MoveL Offs(p0,294.46809999999994,373.47709999999995, 0), v100, z5, tool0;
MoveL Offs(p0,293.07520000000005,371.8112, 0), v100, z5, tool0;
MoveL Offs(p0,291.8875,370.5125, 0), v100, z5, tool0;
MoveL Offs(p0,290.8528,369.5288, 0), v100, z5, tool0;
MoveL Offs(p0,289.9189,368.80789999999996, 0), v100, z5, tool0;
MoveL Offs(p0,289.03360000000004,368.29760000000005, 0), v100, z5, tool0;
MoveL Offs(p0,288.1447,367.94570000000004, 0), v100, z5, tool0;
MoveL Offs(p0,287.2,367.7, 0), v100, z5, tool0;
MoveL Offs(p0,283.18910000000005,366.95770000000005, 0), v100, z5, tool0;
MoveL Offs(p0,279.59280000000007,366.4176000000001, 0), v100, z5, tool0;
MoveL Offs(p0,276.28569999999996,366.08990000000006, 0), v100, z5, tool0;
MoveL Offs(p0,273.1424,365.9848, 0), v100, z5, tool0;
MoveL Offs(p0,270.0375,366.1125, 0), v100, z5, tool0;
MoveL Offs(p0,266.8456,366.4832, 0), v100, z5, tool0;
MoveL Offs(p0,263.4413,367.1071, 0), v100, z5, tool0;
MoveL Offs(p0,259.6992,367.99440000000004, 0), v100, z5, tool0;
MoveL Offs(p0,255.49390000000002,369.1553, 0), v100, z5, tool0;
MoveL Offs(p0,250.7,370.6, 0), v100, z5, tool0;
MoveL Offs(p0,248.47970000000004,371.28720000000004, 0), v100, z5, tool0;
MoveL Offs(p0,246.31760000000008,371.90960000000007, 0), v100, z5, tool0;
MoveL Offs(p0,244.21189999999996,372.4684, 0), v100, z5, tool0;
MoveL Offs(p0,242.16079999999997,372.9648, 0), v100, z5, tool0;
MoveL Offs(p0,240.1625,373.4, 0), v100, z5, tool0;
MoveL Offs(p0,238.2152,373.7752, 0), v100, z5, tool0;
MoveL Offs(p0,236.31709999999998,374.0916, 0), v100, z5, tool0;
MoveL Offs(p0,234.46640000000002,374.35040000000004, 0), v100, z5, tool0;
MoveL Offs(p0,232.66130000000004,374.55280000000005, 0), v100, z5, tool0;
MoveL Offs(p0,230.9,374.7, 0), v100, z5, tool0;
MoveL Offs(p0,222.3,375.3, 0), v100, z5, tool0;
MoveL Offs(p0,221.6,384.4, 0), v100, z5, tool0;
MoveL Offs(p0,221.27370000000005,388.0507, 0), v100, z5, tool0;
MoveL Offs(p0,220.78960000000006,392.02960000000013, 0), v100, z5, tool0;
MoveL Offs(p0,220.1699,396.22690000000006, 0), v100, z5, tool0;
MoveL Offs(p0,219.43680000000003,400.53280000000007, 0), v100, z5, tool0;
MoveL Offs(p0,218.6125,404.8375, 0), v100, z5, tool0;
MoveL Offs(p0,217.7192,409.0312, 0), v100, z5, tool0;
MoveL Offs(p0,216.77910000000003,413.0041, 0), v100, z5, tool0;
MoveL Offs(p0,215.81440000000003,416.6464000000001, 0), v100, z5, tool0;
MoveL Offs(p0,214.8473,419.8483, 0), v100, z5, tool0;
MoveL Offs(p0,213.9,422.5, 0), v100, z5, tool0;
MoveL Offs(p0,213.26730000000003,424.0777, 0), v100, z5, tool0;
MoveL Offs(p0,212.72640000000007,425.3536000000002, 0), v100, z5, tool0;
MoveL Offs(p0,212.2431,426.3619, 0), v100, z5, tool0;
MoveL Offs(p0,211.78320000000002,427.13680000000005, 0), v100, z5, tool0;
MoveL Offs(p0,211.3125,427.7125, 0), v100, z5, tool0;
MoveL Offs(p0,210.7968,428.1232, 0), v100, z5, tool0;
MoveL Offs(p0,210.20190000000002,428.4031, 0), v100, z5, tool0;
MoveL Offs(p0,209.49360000000001,428.5864, 0), v100, z5, tool0;
MoveL Offs(p0,208.6377,428.70730000000003, 0), v100, z5, tool0;
MoveL Offs(p0,207.6,428.8, 0), v100, z5, tool0;
MoveL Offs(p0,203.7,429.1, 0), v100, z5, tool0;
MoveL Offs(p0,204.4,419.3, 0), v100, z5, tool0;
MoveL Offs(p0,205.0,409.5, 0), v100, z5, tool0;
MoveL Offs(p0,201.9,417.0, 0), v100, z5, tool0;
MoveL Offs(p0,200.11920000000003,421.2125000000001, 0), v100, z5, tool0;
MoveL Offs(p0,198.11760000000004,425.7280000000002, 0), v100, z5, tool0;
MoveL Offs(p0,195.9564,430.4235, 0), v100, z5, tool0;
MoveL Offs(p0,193.69680000000002,435.17600000000004, 0), v100, z5, tool0;
MoveL Offs(p0,191.4,439.8625, 0), v100, z5, tool0;
MoveL Offs(p0,189.1272,444.36, 0), v100, z5, tool0;
MoveL Offs(p0,186.9396,448.5455, 0), v100, z5, tool0;
MoveL Offs(p0,184.8984,452.2960000000001, 0), v100, z5, tool0;
MoveL Offs(p0,183.06480000000002,455.48850000000004, 0), v100, z5, tool0;
MoveL Offs(p0,181.5,458.0, 0), v100, z5, tool0;
MoveL Offs(p0,179.79570000000004,460.49500000000006, 0), v100, z5, tool0;
MoveL Offs(p0,178.25760000000002,462.6000000000002, 0), v100, z5, tool0;
MoveL Offs(p0,176.8479,464.34499999999997, 0), v100, z5, tool0;
MoveL Offs(p0,175.5288,465.76000000000005, 0), v100, z5, tool0;
MoveL Offs(p0,174.2625,466.875, 0), v100, z5, tool0;
MoveL Offs(p0,173.0112,467.71999999999997, 0), v100, z5, tool0;
MoveL Offs(p0,171.7371,468.325, 0), v100, z5, tool0;
MoveL Offs(p0,170.4024,468.7200000000001, 0), v100, z5, tool0;
MoveL Offs(p0,168.96930000000003,468.93500000000006, 0), v100, z5, tool0;
MoveL Offs(p0,167.4,469.0, 0), v100, z5, tool0;
MoveL Offs(p0,164.1664,468.7728000000001, 0), v100, z5, tool0;
MoveL Offs(p0,163.7375,468.6125, 0), v100, z5, tool0;
MoveL Offs(p0,163.4256,468.39519999999993, 0), v100, z5, tool0;
MoveL Offs(p0,163.2133,468.11310000000003, 0), v100, z5, tool0;
MoveL Offs(p0,163.0832,467.75840000000005, 0), v100, z5, tool0;
MoveL Offs(p0,163.0179,467.3233, 0), v100, z5, tool0;
MoveL Offs(p0,163.0,466.8, 0), v100, z5, tool0;
MoveL Offs(p0,163.0,466.8, 0), v100, z5, tool0;
MoveJ Offs(p0,173.0,464.5, 10), v100, z1, tool0;
MoveL Offs(p0,174.1694,463.2745000000001, 0), v100, z5, tool0;
MoveL Offs(p0,175.55120000000005,461.56000000000023, 0), v100, z5, tool0;
MoveL Offs(p0,177.1058,459.41949999999997, 0), v100, z5, tool0;
MoveL Offs(p0,178.79360000000003,456.916, 0), v100, z5, tool0;
MoveL Offs(p0,180.575,454.1125, 0), v100, z5, tool0;
MoveL Offs(p0,182.4104,451.07199999999995, 0), v100, z5, tool0;
MoveL Offs(p0,184.2602,447.8575000000001, 0), v100, z5, tool0;
MoveL Offs(p0,186.08480000000003,444.532, 0), v100, z5, tool0;
MoveL Offs(p0,187.8446,441.1585, 0), v100, z5, tool0;
MoveL Offs(p0,189.5,437.8, 0), v100, z5, tool0;
MoveL Offs(p0,191.66320000000002,433.08140000000003, 0), v100, z5, tool0;
MoveL Offs(p0,193.79760000000005,428.1432000000001, 0), v100, z5, tool0;
MoveL Offs(p0,195.85039999999998,423.1318, 0), v100, z5, tool0;
MoveL Offs(p0,197.7688,418.19360000000006, 0), v100, z5, tool0;
MoveL Offs(p0,199.5,413.475, 0), v100, z5, tool0;
MoveL Offs(p0,200.9912,409.1224, 0), v100, z5, tool0;
MoveL Offs(p0,202.1896,405.2822, 0), v100, z5, tool0;
MoveL Offs(p0,203.04240000000001,402.10080000000005, 0), v100, z5, tool0;
MoveL Offs(p0,203.4968,399.7246, 0), v100, z5, tool0;
MoveL Offs(p0,203.5,398.3, 0), v100, z5, tool0;
MoveL Offs(p0,203.88400000000001,396.0856, 0), v100, z5, tool0;
MoveL Offs(p0,204.121,396.0212, 0), v100, z5, tool0;
MoveL Offs(p0,204.4,396.0, 0), v100, z5, tool0;
MoveL Offs(p0,205.57200000000006,396.43520000000007, 0), v100, z5, tool0;
MoveL Offs(p0,206.01099999999997,397.05029999999994, 0), v100, z5, tool0;
MoveL Offs(p0,206.36000000000004,397.9936, 0), v100, z5, tool0;
MoveL Offs(p0,206.625,399.3125, 0), v100, z5, tool0;
MoveL Offs(p0,206.81199999999998,401.0544, 0), v100, z5, tool0;
MoveL Offs(p0,206.927,403.2667, 0), v100, z5, tool0;
MoveL Offs(p0,206.97600000000003,405.9968, 0), v100, z5, tool0;
MoveL Offs(p0,206.965,409.2921, 0), v100, z5, tool0;
MoveL Offs(p0,206.9,413.2, 0), v100, z5, tool0;
MoveL Offs(p0,207.1384,424.5264000000001, 0), v100, z5, tool0;
MoveL Offs(p0,207.4125,425.8625, 0), v100, z5, tool0;
MoveL Offs(p0,207.78560000000002,426.6496, 0), v100, z5, tool0;
MoveL Offs(p0,208.2643,426.91229999999996, 0), v100, z5, tool0;
MoveL Offs(p0,208.85520000000002,426.6752, 0), v100, z5, tool0;
MoveL Offs(p0,209.56490000000002,425.9629, 0), v100, z5, tool0;
MoveL Offs(p0,210.4,424.8, 0), v100, z5, tool0;
MoveL Offs(p0,211.00590000000003,423.62250000000006, 0), v100, z5, tool0;
MoveL Offs(p0,211.67120000000006,421.8840000000001, 0), v100, z5, tool0;
MoveL Offs(p0,212.37730000000002,419.66549999999995, 0), v100, z5, tool0;
MoveL Offs(p0,213.1056,417.04799999999994, 0), v100, z5, tool0;
MoveL Offs(p0,213.8375,414.1125, 0), v100, z5, tool0;
MoveL Offs(p0,214.55440000000004,410.93999999999994, 0), v100, z5, tool0;
MoveL Offs(p0,215.2377,407.6115, 0), v100, z5, tool0;
MoveL Offs(p0,215.86880000000002,404.208, 0), v100, z5, tool0;
MoveL Offs(p0,216.4291,400.81050000000005, 0), v100, z5, tool0;
MoveL Offs(p0,216.9,397.5, 0), v100, z5, tool0;
MoveL Offs(p0,217.40370000000001,393.5277000000001, 0), v100, z5, tool0;
MoveL Offs(p0,217.83360000000008,389.8536000000001, 0), v100, z5, tool0;
MoveL Offs(p0,218.18789999999998,386.51189999999997, 0), v100, z5, tool0;
MoveL Offs(p0,218.46480000000003,383.5368, 0), v100, z5, tool0;
MoveL Offs(p0,218.6625,380.9625, 0), v100, z5, tool0;
MoveL Offs(p0,218.7792,378.8232, 0), v100, z5, tool0;
MoveL Offs(p0,218.8131,377.1531, 0), v100, z5, tool0;
MoveL Offs(p0,218.7624,375.98640000000006, 0), v100, z5, tool0;
MoveL Offs(p0,218.6253,375.3573, 0), v100, z5, tool0;
MoveL Offs(p0,218.4,375.3, 0), v100, z5, tool0;
MoveL Offs(p0,218.07510000000002,375.6689, 0), v100, z5, tool0;
MoveL Offs(p0,217.42080000000004,376.45120000000014, 0), v100, z5, tool0;
MoveL Offs(p0,216.46769999999998,377.6103, 0), v100, z5, tool0;
MoveL Offs(p0,215.24640000000005,379.10960000000006, 0), v100, z5, tool0;
MoveL Offs(p0,213.7875,380.9125, 0), v100, z5, tool0;
MoveL Offs(p0,212.1216,382.9824, 0), v100, z5, tool0;
MoveL Offs(p0,210.2793,385.28270000000003, 0), v100, z5, tool0;
MoveL Offs(p0,208.29120000000003,387.77680000000004, 0), v100, z5, tool0;
MoveL Offs(p0,206.18789999999998,390.4281, 0), v100, z5, tool0;
MoveL Offs(p0,204.0,393.2, 0), v100, z5, tool0;
MoveL Offs(p0,201.8005,396.0019000000001, 0), v100, z5, tool0;
MoveL Offs(p0,199.66400000000004,398.68320000000006, 0), v100, z5, tool0;
MoveL Offs(p0,197.62349999999998,401.2073, 0), v100, z5, tool0;
MoveL Offs(p0,195.71200000000002,403.5376, 0), v100, z5, tool0;
MoveL Offs(p0,193.9625,405.6375, 0), v100, z5, tool0;
MoveL Offs(p0,192.40800000000002,407.4704, 0), v100, z5, tool0;
MoveL Offs(p0,191.0815,408.99969999999996, 0), v100, z5, tool0;
MoveL Offs(p0,190.01600000000002,410.1888, 0), v100, z5, tool0;
MoveL Offs(p0,189.24450000000002,411.00110000000006, 0), v100, z5, tool0;
MoveL Offs(p0,188.8,411.4, 0), v100, z5, tool0;
MoveL Offs(p0,188.18900000000002,411.6944, 0), v100, z5, tool0;
MoveL Offs(p0,187.56000000000003,411.85920000000004, 0), v100, z5, tool0;
MoveL Offs(p0,186.919,411.8968, 0), v100, z5, tool0;
MoveL Offs(p0,186.27200000000002,411.80959999999993, 0), v100, z5, tool0;
MoveL Offs(p0,185.625,411.6, 0), v100, z5, tool0;
MoveL Offs(p0,184.35499999999996,410.8232, 0), v100, z5, tool0;
MoveL Offs(p0,183.744,410.2608, 0), v100, z5, tool0;
MoveL Offs(p0,183.157,409.5856, 0), v100, z5, tool0;
MoveL Offs(p0,182.6,408.8, 0), v100, z5, tool0;
MoveL Offs(p0,182.29110000000003,408.22150000000005, 0), v100, z5, tool0;
MoveL Offs(p0,182.14480000000006,407.54400000000015, 0), v100, z5, tool0;
MoveL Offs(p0,182.2517,406.55449999999996, 0), v100, z5, tool0;
MoveL Offs(p0,183.5875,402.7875, 0), v100, z5, tool0;
MoveL Offs(p0,184.9976,399.58399999999995, 0), v100, z5, tool0;
MoveL Offs(p0,187.0233,395.2165, 0), v100, z5, tool0;
MoveL Offs(p0,189.7552,389.47200000000004, 0), v100, z5, tool0;
MoveL Offs(p0,193.28390000000002,382.1375, 0), v100, z5, tool0;
MoveL Offs(p0,197.7,373.0, 0), v100, z5, tool0;
MoveL Offs(p0,199.66400000000002,368.88100000000014, 0), v100, z5, tool0;
MoveL Offs(p0,201.52000000000007,364.96000000000004, 0), v100, z5, tool0;
MoveL Offs(p0,203.244,361.29100000000005, 0), v100, z5, tool0;
MoveL Offs(p0,204.81200000000004,357.928, 0), v100, z5, tool0;
MoveL Offs(p0,206.2,354.925, 0), v100, z5, tool0;
MoveL Offs(p0,207.38400000000001,352.33599999999996, 0), v100, z5, tool0;
MoveL Offs(p0,208.34,350.21500000000003, 0), v100, z5, tool0;
MoveL Offs(p0,209.04400000000004,348.61600000000004, 0), v100, z5, tool0;
MoveL Offs(p0,209.47200000000004,347.593, 0), v100, z5, tool0;
MoveL Offs(p0,209.6,347.2, 0), v100, z5, tool0;
MoveL Offs(p0,208.92859999999996,347.4196, 0), v100, z5, tool0;
MoveL Offs(p0,208.5152,347.6512000000001, 0), v100, z5, tool0;
MoveL Offs(p0,208.025,347.95, 0), v100, z5, tool0;
MoveL Offs(p0,207.46880000000002,348.3088, 0), v100, z5, tool0;
MoveL Offs(p0,206.85739999999996,348.7204, 0), v100, z5, tool0;
MoveL Offs(p0,206.2016,349.17760000000004, 0), v100, z5, tool0;
MoveL Offs(p0,205.51220000000004,349.67320000000007, 0), v100, z5, tool0;
MoveL Offs(p0,204.8,350.2, 0), v100, z5, tool0;
MoveL Offs(p0,203.59520000000003,351.0874, 0), v100, z5, tool0;
MoveL Offs(p0,202.32560000000007,351.9472000000001, 0), v100, z5, tool0;
MoveL Offs(p0,200.9984,352.7758, 0), v100, z5, tool0;
MoveL Offs(p0,199.62080000000003,353.5696, 0), v100, z5, tool0;
MoveL Offs(p0,198.2,354.325, 0), v100, z5, tool0;
MoveL Offs(p0,196.7432,355.0384, 0), v100, z5, tool0;
MoveL Offs(p0,195.2576,355.70619999999997, 0), v100, z5, tool0;
MoveL Offs(p0,193.75040000000004,356.3248, 0), v100, z5, tool0;
MoveL Offs(p0,192.2288,356.8906, 0), v100, z5, tool0;
MoveL Offs(p0,190.7,357.4, 0), v100, z5, tool0;
MoveL Offs(p0,190.04080000000005,357.8960000000001, 0), v100, z5, tool0;
MoveL Offs(p0,189.63619999999997,358.3585, 0), v100, z5, tool0;
MoveL Offs(p0,189.1944,358.944, 0), v100, z5, tool0;
MoveL Offs(p0,188.725,359.6375, 0), v100, z5, tool0;
MoveL Offs(p0,188.2376,360.424, 0), v100, z5, tool0;
MoveL Offs(p0,187.7418,361.2885, 0), v100, z5, tool0;
MoveL Offs(p0,187.24720000000002,362.216, 0), v100, z5, tool0;
MoveL Offs(p0,186.7634,363.1915, 0), v100, z5, tool0;
MoveL Offs(p0,186.3,364.2, 0), v100, z5, tool0;
MoveL Offs(p0,185.02380000000002,367.0821, 0), v100, z5, tool0;
MoveL Offs(p0,183.65040000000005,370.0368000000001, 0), v100, z5, tool0;
MoveL Offs(p0,182.1726,373.07669999999996, 0), v100, z5, tool0;
MoveL Offs(p0,180.58319999999998,376.2144, 0), v100, z5, tool0;
MoveL Offs(p0,178.875,379.4625, 0), v100, z5, tool0;
MoveL Offs(p0,177.04080000000002,382.83360000000005, 0), v100, z5, tool0;
MoveL Offs(p0,175.0734,386.3403, 0), v100, z5, tool0;
MoveL Offs(p0,172.96560000000002,389.9952, 0), v100, z5, tool0;
MoveL Offs(p0,170.71020000000001,393.81090000000006, 0), v100, z5, tool0;
MoveL Offs(p0,168.3,397.8, 0), v100, z5, tool0;
MoveL Offs(p0,167.0781,399.8056, 0), v100, z5, tool0;
MoveL Offs(p0,165.94080000000005,401.7248000000001, 0), v100, z5, tool0;
MoveL Offs(p0,164.90069999999997,403.5312, 0), v100, z5, tool0;
MoveL Offs(p0,163.9704,405.19840000000005, 0), v100, z5, tool0;
MoveL Offs(p0,163.1625,406.7, 0), v100, z5, tool0;
MoveL Offs(p0,162.48960000000002,408.0096, 0), v100, z5, tool0;
MoveL Offs(p0,161.9643,409.1008, 0), v100, z5, tool0;
MoveL Offs(p0,161.59920000000002,409.94719999999995, 0), v100, z5, tool0;
MoveL Offs(p0,161.4069,410.5224, 0), v100, z5, tool0;
MoveL Offs(p0,161.4,410.8, 0), v100, z5, tool0;
MoveL Offs(p0,163.78140000000002,410.3509, 0), v100, z5, tool0;
MoveL Offs(p0,165.0688,409.7888000000001, 0), v100, z5, tool0;
MoveL Offs(p0,166.475,409.0875, 0), v100, z5, tool0;
MoveL Offs(p0,167.9232,408.2872, 0), v100, z5, tool0;
MoveL Offs(p0,169.3366,407.4281, 0), v100, z5, tool0;
MoveL Offs(p0,170.6384,406.5504, 0), v100, z5, tool0;
MoveL Offs(p0,171.7518,405.6943, 0), v100, z5, tool0;
MoveL Offs(p0,172.6,404.9, 0), v100, z5, tool0;
MoveL Offs(p0,172.97840000000002,404.47540000000004, 0), v100, z5, tool0;
MoveL Offs(p0,173.2752,404.0952000000001, 0), v100, z5, tool0;
MoveL Offs(p0,173.4928,403.7498, 0), v100, z5, tool0;
MoveL Offs(p0,173.63360000000003,403.42960000000005, 0), v100, z5, tool0;
MoveL Offs(p0,173.7,403.125, 0), v100, z5, tool0;
MoveL Offs(p0,173.6944,402.82640000000004, 0), v100, z5, tool0;
MoveL Offs(p0,173.6192,402.5242, 0), v100, z5, tool0;
MoveL Offs(p0,173.4768,402.2088, 0), v100, z5, tool0;
MoveL Offs(p0,173.2696,401.8706, 0), v100, z5, tool0;
MoveL Offs(p0,173.0,401.5, 0), v100, z5, tool0;
MoveL Offs(p0,172.70970000000003,401.1421, 0), v100, z5, tool0;
MoveL Offs(p0,172.50160000000005,400.8448000000001, 0), v100, z5, tool0;
MoveL Offs(p0,172.37989999999996,400.6027, 0), v100, z5, tool0;
MoveL Offs(p0,172.34880000000004,400.41040000000004, 0), v100, z5, tool0;
MoveL Offs(p0,172.4125,400.2625, 0), v100, z5, tool0;
MoveL Offs(p0,172.5752,400.1536, 0), v100, z5, tool0;
MoveL Offs(p0,173.2144,400.0312, 0), v100, z5, tool0;
MoveL Offs(p0,173.6993,400.00690000000003, 0), v100, z5, tool0;
MoveL Offs(p0,174.3,400.0, 0), v100, z5, tool0;
MoveL Offs(p0,176.0456,400.3296, 0), v100, z5, tool0;
MoveL Offs(p0,176.3875,400.5125, 0), v100, z5, tool0;
MoveL Offs(p0,176.6904,400.7344, 0), v100, z5, tool0;
MoveL Offs(p0,176.95369999999997,400.9947, 0), v100, z5, tool0;
MoveL Offs(p0,177.17680000000001,401.29280000000006, 0), v100, z5, tool0;
MoveL Offs(p0,177.3591,401.6281, 0), v100, z5, tool0;
MoveL Offs(p0,177.5,402.0, 0), v100, z5, tool0;
MoveL Offs(p0,177.74540000000002,404.81690000000003, 0), v100, z5, tool0;
MoveL Offs(p0,176.7278,415.86629999999997, 0), v100, z5, tool0;
MoveL Offs(p0,175.63760000000002,423.1616, 0), v100, z5, tool0;
MoveL Offs(p0,174.275,431.0125, 0), v100, z5, tool0;
MoveL Offs(p0,172.72639999999998,438.9504, 0), v100, z5, tool0;
MoveL Offs(p0,171.07819999999998,446.5067, 0), v100, z5, tool0;
MoveL Offs(p0,169.41680000000002,453.2128000000001, 0), v100, z5, tool0;
MoveL Offs(p0,167.8286,458.6001, 0), v100, z5, tool0;
MoveL Offs(p0,166.4,462.2, 0), v100, z5, tool0;
MoveL Offs(p0,166.1723,462.6817000000001, 0), v100, z5, tool0;
MoveL Offs(p0,165.97040000000004,463.1616000000001, 0), v100, z5, tool0;
MoveL Offs(p0,165.79609999999997,463.6319, 0), v100, z5, tool0;
MoveL Offs(p0,165.65120000000002,464.0848, 0), v100, z5, tool0;
MoveL Offs(p0,165.5375,464.5125, 0), v100, z5, tool0;
MoveL Offs(p0,165.4568,464.9072, 0), v100, z5, tool0;
MoveL Offs(p0,165.41090000000003,465.2611, 0), v100, z5, tool0;
MoveL Offs(p0,165.4016,465.56640000000004, 0), v100, z5, tool0;
MoveL Offs(p0,165.4307,465.81530000000004, 0), v100, z5, tool0;
MoveL Offs(p0,165.5,466.0, 0), v100, z5, tool0;
MoveL Offs(p0,165.872,466.3495000000001, 0), v100, z5, tool0;
MoveL Offs(p0,166.42400000000004,466.56400000000014, 0), v100, z5, tool0;
MoveL Offs(p0,167.11999999999998,466.6525, 0), v100, z5, tool0;
MoveL Offs(p0,167.924,466.62399999999997, 0), v100, z5, tool0;
MoveL Offs(p0,168.8,466.4875, 0), v100, z5, tool0;
MoveL Offs(p0,169.712,466.25199999999995, 0), v100, z5, tool0;
MoveL Offs(p0,171.5,465.5200000000001, 0), v100, z5, tool0;
MoveL Offs(p0,172.304,465.0415, 0), v100, z5, tool0;
MoveL Offs(p0,173.0,464.5, 0), v100, z5, tool0;
MoveL Offs(p0,173.0,464.5, 0), v100, z5, tool0;
MoveJ Offs(p0,131.0,391.0, 10), v100, z1, tool0;
MoveL Offs(p0,134.57830000000004,388.8518, 0), v100, z5, tool0;
MoveL Offs(p0,137.85840000000002,386.7984000000001, 0), v100, z5, tool0;
MoveL Offs(p0,140.81810000000002,384.85659999999996, 0), v100, z5, tool0;
MoveL Offs(p0,143.43520000000004,383.0432, 0), v100, z5, tool0;
MoveL Offs(p0,145.6875,381.375, 0), v100, z5, tool0;
MoveL Offs(p0,147.5528,379.8688, 0), v100, z5, tool0;
MoveL Offs(p0,149.00889999999998,378.54139999999995, 0), v100, z5, tool0;
MoveL Offs(p0,150.03360000000004,377.40960000000007, 0), v100, z5, tool0;
MoveL Offs(p0,150.6047,376.4902, 0), v100, z5, tool0;
MoveL Offs(p0,150.7,375.8, 0), v100, z5, tool0;
MoveL Offs(p0,151.0,374.0, 0), v100, z5, tool0;
MoveL Offs(p0,151.93920000000006,374.2992000000001, 0), v100, z5, tool0;
MoveL Offs(p0,152.2618,374.68580000000003, 0), v100, z5, tool0;
MoveL Offs(p0,152.48960000000002,375.24160000000006, 0), v100, z5, tool0;
MoveL Offs(p0,152.625,375.975, 0), v100, z5, tool0;
MoveL Offs(p0,152.6704,376.89439999999996, 0), v100, z5, tool0;
MoveL Offs(p0,152.62820000000002,378.0082, 0), v100, z5, tool0;
MoveL Offs(p0,152.50080000000003,379.32480000000004, 0), v100, z5, tool0;
MoveL Offs(p0,152.29059999999998,380.85260000000005, 0), v100, z5, tool0;
MoveL Offs(p0,152.0,382.6, 0), v100, z5, tool0;
MoveL Offs(p0,151.63040000000007,384.6920000000001, 0), v100, z5, tool0;
MoveL Offs(p0,151.4861,385.66450000000003, 0), v100, z5, tool0;
MoveL Offs(p0,151.3712,386.56800000000004, 0), v100, z5, tool0;
MoveL Offs(p0,151.2875,387.3875, 0), v100, z5, tool0;
MoveL Offs(p0,151.23679999999996,388.108, 0), v100, z5, tool0;
MoveL Offs(p0,151.22089999999997,388.71449999999993, 0), v100, z5, tool0;
MoveL Offs(p0,151.2416,389.19200000000006, 0), v100, z5, tool0;
MoveL Offs(p0,151.3007,389.5255, 0), v100, z5, tool0;
MoveL Offs(p0,151.4,389.7, 0), v100, z5, tool0;
MoveL Offs(p0,153.60960000000006,388.6432000000001, 0), v100, z5, tool0;
MoveL Offs(p0,155.5094,386.83079999999995, 0), v100, z5, tool0;
MoveL Offs(p0,157.77280000000002,384.36560000000003, 0), v100, z5, tool0;
MoveL Offs(p0,160.275,381.4, 0), v100, z5, tool0;
MoveL Offs(p0,162.8912,378.08639999999997, 0), v100, z5, tool0;
MoveL Offs(p0,165.4966,374.5772, 0), v100, z5, tool0;
MoveL Offs(p0,167.96640000000002,371.0248, 0), v100, z5, tool0;
MoveL Offs(p0,170.1758,367.5816, 0), v100, z5, tool0;
MoveL Offs(p0,172.0,364.4, 0), v100, z5, tool0;
MoveL Offs(p0,174.3,360.2, 0), v100, z5, tool0;
MoveL Offs(p0,166.4,352.6, 0), v100, z5, tool0;
MoveL Offs(p0,164.95190000000002,351.2269, 0), v100, z5, tool0;
MoveL Offs(p0,163.61120000000005,349.99120000000005, 0), v100, z5, tool0;
MoveL Offs(p0,162.3833,348.89829999999995, 0), v100, z5, tool0;
MoveL Offs(p0,161.27360000000002,347.95360000000005, 0), v100, z5, tool0;
MoveL Offs(p0,160.2875,347.1625, 0), v100, z5, tool0;
MoveL Offs(p0,159.4304,346.5304, 0), v100, z5, tool0;
MoveL Offs(p0,158.7077,346.0627, 0), v100, z5, tool0;
MoveL Offs(p0,158.1248,345.76480000000004, 0), v100, z5, tool0;
MoveL Offs(p0,157.68710000000002,345.6421, 0), v100, z5, tool0;
MoveL Offs(p0,157.4,345.7, 0), v100, z5, tool0;
MoveL Offs(p0,157.06470000000002,345.91020000000003, 0), v100, z5, tool0;
MoveL Offs(p0,156.49360000000007,346.28960000000006, 0), v100, z5, tool0;
MoveL Offs(p0,155.7089,346.8214, 0), v100, z5, tool0;
MoveL Offs(p0,154.7328,347.48879999999997, 0), v100, z5, tool0;
MoveL Offs(p0,153.5875,348.275, 0), v100, z5, tool0;
MoveL Offs(p0,152.29519999999997,349.1632, 0), v100, z5, tool0;
MoveL Offs(p0,150.8781,350.1366, 0), v100, z5, tool0;
MoveL Offs(p0,149.35840000000002,351.1784, 0), v100, z5, tool0;
MoveL Offs(p0,147.75830000000002,352.27180000000004, 0), v100, z5, tool0;
MoveL Offs(p0,146.1,353.4, 0), v100, z5, tool0;
MoveL Offs(p0,144.4807,354.50120000000004, 0), v100, z5, tool0;
MoveL Offs(p0,142.93760000000003,355.57360000000006, 0), v100, z5, tool0;
MoveL Offs(p0,141.4929,356.6004, 0), v100, z5, tool0;
MoveL Offs(p0,140.1688,357.5648, 0), v100, z5, tool0;
MoveL Offs(p0,138.9875,358.45, 0), v100, z5, tool0;
MoveL Offs(p0,137.9712,359.2392, 0), v100, z5, tool0;
MoveL Offs(p0,137.14209999999997,359.9156, 0), v100, z5, tool0;
MoveL Offs(p0,136.5224,360.4624, 0), v100, z5, tool0;
MoveL Offs(p0,136.1343,360.8628, 0), v100, z5, tool0;
MoveL Offs(p0,136.0,361.1, 0), v100, z5, tool0;
MoveL Offs(p0,136.20480000000003,361.38560000000007, 0), v100, z5, tool0;
MoveL Offs(p0,136.44819999999999,361.5149, 0), v100, z5, tool0;
MoveL Offs(p0,136.7744,361.63280000000003, 0), v100, z5, tool0;
MoveL Offs(p0,137.175,361.7375, 0), v100, z5, tool0;
MoveL Offs(p0,137.64159999999998,361.8272, 0), v100, z5, tool0;
MoveL Offs(p0,138.1658,361.9001, 0), v100, z5, tool0;
MoveL Offs(p0,138.73920000000004,361.9544, 0), v100, z5, tool0;
MoveL Offs(p0,139.35340000000002,361.98830000000004, 0), v100, z5, tool0;
MoveL Offs(p0,140.0,362.0, 0), v100, z5, tool0;
MoveL Offs(p0,142.772,361.6922, 0), v100, z5, tool0;
MoveL Offs(p0,143.37600000000003,361.4784, 0), v100, z5, tool0;
MoveL Offs(p0,143.8,361.225, 0), v100, z5, tool0;
MoveL Offs(p0,144.03199999999998,360.9416, 0), v100, z5, tool0;
MoveL Offs(p0,144.06,360.63779999999997, 0), v100, z5, tool0;
MoveL Offs(p0,143.872,360.3232, 0), v100, z5, tool0;
MoveL Offs(p0,143.45600000000002,360.0074, 0), v100, z5, tool0;
MoveL Offs(p0,142.8,359.7, 0), v100, z5, tool0;
MoveL Offs(p0,142.32569999999998,359.43809999999996, 0), v100, z5, tool0;
MoveL Offs(p0,142.2784,359.3592, 0), v100, z5, tool0;
MoveL Offs(p0,142.2875,359.2875, 0), v100, z5, tool0;
MoveL Offs(p0,142.35359999999997,359.2248, 0), v100, z5, tool0;
MoveL Offs(p0,142.4773,359.17289999999997, 0), v100, z5, tool0;
MoveL Offs(p0,143.2,359.1, 0), v100, z5, tool0;
MoveL Offs(p0,144.9073,359.4636, 0), v100, z5, tool0;
MoveL Offs(p0,145.23360000000002,359.7832, 0), v100, z5, tool0;
MoveL Offs(p0,145.4375,360.2, 0), v100, z5, tool0;
MoveL Offs(p0,145.51839999999999,360.71279999999996, 0), v100, z5, tool0;
MoveL Offs(p0,145.4757,361.32039999999995, 0), v100, z5, tool0;
MoveL Offs(p0,145.30880000000002,362.02160000000003, 0), v100, z5, tool0;
MoveL Offs(p0,145.01710000000003,362.81520000000006, 0), v100, z5, tool0;
MoveL Offs(p0,144.6,363.7, 0), v100, z5, tool0;
MoveL Offs(p0,144.19400000000002,364.33000000000004, 0), v100, z5, tool0;
MoveL Offs(p0,143.47600000000003,365.29600000000005, 0), v100, z5, tool0;
MoveL Offs(p0,142.476,366.562, 0), v100, z5, tool0;
MoveL Offs(p0,141.22400000000002,368.09200000000004, 0), v100, z5, tool0;
MoveL Offs(p0,139.75,369.85, 0), v100, z5, tool0;
MoveL Offs(p0,138.084,371.79999999999995, 0), v100, z5, tool0;
MoveL Offs(p0,136.256,373.906, 0), v100, z5, tool0;
MoveL Offs(p0,134.296,376.132, 0), v100, z5, tool0;
MoveL Offs(p0,132.234,378.442, 0), v100, z5, tool0;
MoveL Offs(p0,130.1,380.8, 0), v100, z5, tool0;
MoveL Offs(p0,127.98949999999999,383.1318, 0), v100, z5, tool0;
MoveL Offs(p0,125.99600000000002,385.3664000000001, 0), v100, z5, tool0;
MoveL Offs(p0,124.14649999999999,387.47259999999994, 0), v100, z5, tool0;
MoveL Offs(p0,122.468,389.41920000000005, 0), v100, z5, tool0;
MoveL Offs(p0,120.9875,391.175, 0), v100, z5, tool0;
MoveL Offs(p0,119.732,392.7088, 0), v100, z5, tool0;
MoveL Offs(p0,118.72849999999998,393.98940000000005, 0), v100, z5, tool0;
MoveL Offs(p0,118.00399999999999,394.98560000000003, 0), v100, z5, tool0;
MoveL Offs(p0,117.5855,395.6662, 0), v100, z5, tool0;
MoveL Offs(p0,117.5,396.0, 0), v100, z5, tool0;
MoveL Offs(p0,117.8672,396.2596, 0), v100, z5, tool0;
MoveL Offs(p0,118.52960000000003,396.32480000000015, 0), v100, z5, tool0;
MoveL Offs(p0,119.45840000000003,396.2052, 0), v100, z5, tool0;
MoveL Offs(p0,122.0,395.45, 0), v100, z5, tool0;
MoveL Offs(p0,123.55520000000001,394.83360000000005, 0), v100, z5, tool0;
MoveL Offs(p0,125.2616,394.07079999999996, 0), v100, z5, tool0;
MoveL Offs(p0,127.0904,393.17120000000006, 0), v100, z5, tool0;
MoveL Offs(p0,129.01280000000003,392.1444, 0), v100, z5, tool0;
MoveL Offs(p0,131.0,391.0, 0), v100, z5, tool0;
MoveL Offs(p0,131.0,391.0, 0), v100, z5, tool0;
MoveJ Offs(p0,427.0,387.6, 10), v100, z1, tool0;
MoveL Offs(p0,426.6328,385.30409999999995, 0), v100, z5, tool0;
MoveL Offs(p0,426.2576,384.66720000000004, 0), v100, z5, tool0;
MoveL Offs(p0,425.7,384.0375, 0), v100, z5, tool0;
MoveL Offs(p0,424.92639999999994,383.3808, 0), v100, z5, tool0;
MoveL Offs(p0,423.9032,382.6629, 0), v100, z5, tool0;
MoveL Offs(p0,422.5968000000001,381.84960000000007, 0), v100, z5, tool0;
MoveL Offs(p0,420.9736,380.9067, 0), v100, z5, tool0;
MoveL Offs(p0,419.0,379.8, 0), v100, z5, tool0;
MoveL Offs(p0,417.89930000000004,379.1782, 0), v100, z5, tool0;
MoveL Offs(p0,416.77040000000017,378.5216000000001, 0), v100, z5, tool0;
MoveL Offs(p0,415.6331,377.8434, 0), v100, z5, tool0;
MoveL Offs(p0,414.5072,377.15680000000003, 0), v100, z5, tool0;
MoveL Offs(p0,413.4125,376.475, 0), v100, z5, tool0;
MoveL Offs(p0,412.3688,375.8112, 0), v100, z5, tool0;
MoveL Offs(p0,411.3959,375.1786, 0), v100, z5, tool0;
MoveL Offs(p0,410.51360000000005,374.59040000000005, 0), v100, z5, tool0;
MoveL Offs(p0,409.74170000000004,374.0598, 0), v100, z5, tool0;
MoveL Offs(p0,409.1,373.6, 0), v100, z5, tool0;
MoveL Offs(p0,408.5314,373.19570000000004, 0), v100, z5, tool0;
MoveL Offs(p0,407.9712000000001,372.8256000000001, 0), v100, z5, tool0;
MoveL Offs(p0,407.42780000000005,372.49389999999994, 0), v100, z5, tool0;
MoveL Offs(p0,406.90960000000007,372.20480000000003, 0), v100, z5, tool0;
MoveL Offs(p0,406.425,371.9625, 0), v100, z5, tool0;
MoveL Offs(p0,405.9824,371.7712, 0), v100, z5, tool0;
MoveL Offs(p0,405.5902,371.6351000000001, 0), v100, z5, tool0;
MoveL Offs(p0,405.2568,371.5584, 0), v100, z5, tool0;
MoveL Offs(p0,404.9906,371.54530000000005, 0), v100, z5, tool0;
MoveL Offs(p0,404.8,371.6, 0), v100, z5, tool0;
MoveL Offs(p0,404.179,371.3408, 0), v100, z5, tool0;
MoveL Offs(p0,404.2,371.2, 0), v100, z5, tool0;
MoveL Offs(p0,403.92080000000004,370.55920000000015, 0), v100, z5, tool0;
MoveL Offs(p0,403.50519999999995,370.0498, 0), v100, z5, tool0;
MoveL Offs(p0,402.9264,369.4336, 0), v100, z5, tool0;
MoveL Offs(p0,402.2,368.725, 0), v100, z5, tool0;
MoveL Offs(p0,401.3416,367.93839999999994, 0), v100, z5, tool0;
MoveL Offs(p0,400.36679999999996,367.0882, 0), v100, z5, tool0;
MoveL Offs(p0,399.2912,366.1888, 0), v100, z5, tool0;
MoveL Offs(p0,398.1304,365.25460000000004, 0), v100, z5, tool0;
MoveL Offs(p0,396.9,364.3, 0), v100, z5, tool0;
MoveL Offs(p0,394.46110000000004,362.4155, 0), v100, z5, tool0;
MoveL Offs(p0,392.0768000000001,360.5520000000001, 0), v100, z5, tool0;
MoveL Offs(p0,389.7657,358.7245, 0), v100, z5, tool0;
MoveL Offs(p0,387.54640000000006,356.94800000000004, 0), v100, z5, tool0;
MoveL Offs(p0,385.4375,355.2375, 0), v100, z5, tool0;
MoveL Offs(p0,383.4576,353.60800000000006, 0), v100, z5, tool0;
MoveL Offs(p0,381.6253,352.0745, 0), v100, z5, tool0;
MoveL Offs(p0,379.95920000000007,350.65200000000004, 0), v100, z5, tool0;
MoveL Offs(p0,378.47790000000003,349.3555, 0), v100, z5, tool0;
MoveL Offs(p0,377.2,348.2, 0), v100, z5, tool0;
MoveL Offs(p0,376.61000000000007,347.70760000000007, 0), v100, z5, tool0;
MoveL Offs(p0,376.0920000000001,347.3088000000001, 0), v100, z5, tool0;
MoveL Offs(p0,375.63399999999996,347.00120000000004, 0), v100, z5, tool0;
MoveL Offs(p0,375.22400000000005,346.7824, 0), v100, z5, tool0;
MoveL Offs(p0,374.85,346.65, 0), v100, z5, tool0;
MoveL Offs(p0,374.5,346.60159999999996, 0), v100, z5, tool0;
MoveL Offs(p0,374.162,346.6347999999999, 0), v100, z5, tool0;
MoveL Offs(p0,373.824,346.7472000000001, 0), v100, z5, tool0;
MoveL Offs(p0,373.47400000000005,346.9364, 0), v100, z5, tool0;
MoveL Offs(p0,373.1,347.2, 0), v100, z5, tool0;
MoveL Offs(p0,372.72170000000006,347.49660000000006, 0), v100, z5, tool0;
MoveL Offs(p0,372.4256000000001,347.7248000000001, 0), v100, z5, tool0;
MoveL Offs(p0,372.2099,347.88219999999995, 0), v100, z5, tool0;
MoveL Offs(p0,372.07280000000003,347.9664000000001, 0), v100, z5, tool0;
MoveL Offs(p0,372.0125,347.975, 0), v100, z5, tool0;
MoveL Offs(p0,372.0272,347.90559999999994, 0), v100, z5, tool0;
MoveL Offs(p0,372.1151,347.7558, 0), v100, z5, tool0;
MoveL Offs(p0,372.27440000000007,347.52320000000003, 0), v100, z5, tool0;
MoveL Offs(p0,372.8,346.8, 0), v100, z5, tool0;
MoveL Offs(p0,373.0791000000001,346.39390000000003, 0), v100, z5, tool0;
MoveL Offs(p0,373.2448000000001,345.99920000000014, 0), v100, z5, tool0;
MoveL Offs(p0,373.2797,345.59129999999993, 0), v100, z5, tool0;
MoveL Offs(p0,373.16639999999995,345.14559999999994, 0), v100, z5, tool0;
MoveL Offs(p0,372.42560000000003,344.04239999999993, 0), v100, z5, tool0;
MoveL Offs(p0,371.76329999999996,343.3357, 0), v100, z5, tool0;
MoveL Offs(p0,370.88320000000004,342.4928000000001, 0), v100, z5, tool0;
MoveL Offs(p0,369.7679,341.4891, 0), v100, z5, tool0;
MoveL Offs(p0,368.4,340.3, 0), v100, z5, tool0;
MoveL Offs(p0,367.47810000000004,339.5368, 0), v100, z5, tool0;
MoveL Offs(p0,366.58080000000007,338.8144000000001, 0), v100, z5, tool0;
MoveL Offs(p0,365.72069999999997,338.1436, 0), v100, z5, tool0;
MoveL Offs(p0,364.9104000000001,337.5352000000001, 0), v100, z5, tool0;
MoveL Offs(p0,364.1625,337.0, 0), v100, z5, tool0;
MoveL Offs(p0,363.4896,336.5488, 0), v100, z5, tool0;
MoveL Offs(p0,362.9043,336.1924, 0), v100, z5, tool0;
MoveL Offs(p0,362.4192,335.9416, 0), v100, z5, tool0;
MoveL Offs(p0,362.0469,335.8072, 0), v100, z5, tool0;
MoveL Offs(p0,361.8,335.8, 0), v100, z5, tool0;
MoveL Offs(p0,361.2596,335.569, 0), v100, z5, tool0;
MoveL Offs(p0,361.27840000000003,335.46400000000006, 0), v100, z5, tool0;
MoveL Offs(p0,361.3248,335.341, 0), v100, z5, tool0;
MoveL Offs(p0,361.4,335.2, 0), v100, z5, tool0;
MoveL Offs(p0,360.89239999999995,334.06149999999997, 0), v100, z5, tool0;
MoveL Offs(p0,360.4128,333.41600000000005, 0), v100, z5, tool0;
MoveL Offs(p0,359.8,332.6625, 0), v100, z5, tool0;
MoveL Offs(p0,359.0672,331.8159999999999, 0), v100, z5, tool0;
MoveL Offs(p0,358.2276,330.8915, 0), v100, z5, tool0;
MoveL Offs(p0,357.29440000000005,329.904, 0), v100, z5, tool0;
MoveL Offs(p0,356.2808,328.86850000000004, 0), v100, z5, tool0;
MoveL Offs(p0,355.2,327.8, 0), v100, z5, tool0;
MoveL Offs(p0,354.04330000000004,326.66740000000004, 0), v100, z5, tool0;
MoveL Offs(p0,352.81040000000013,325.4472000000001, 0), v100, z5, tool0;
MoveL Offs(p0,351.5271,324.1658, 0), v100, z5, tool0;
MoveL Offs(p0,350.2192,322.84960000000007, 0), v100, z5, tool0;
MoveL Offs(p0,348.9125,321.525, 0), v100, z5, tool0;
MoveL Offs(p0,347.6328,320.2184, 0), v100, z5, tool0;
MoveL Offs(p0,346.4059,318.95619999999997, 0), v100, z5, tool0;
MoveL Offs(p0,345.2576,317.76480000000004, 0), v100, z5, tool0;
MoveL Offs(p0,344.21369999999996,316.67060000000004, 0), v100, z5, tool0;
MoveL Offs(p0,343.3,315.7, 0), v100, z5, tool0;
MoveL Offs(p0,342.47100000000006,314.79580000000004, 0), v100, z5, tool0;
MoveL Offs(p0,341.6720000000001,313.95040000000006, 0), v100, z5, tool0;
MoveL Offs(p0,340.915,313.17459999999994, 0), v100, z5, tool0;
MoveL Offs(p0,340.21200000000005,312.47920000000005, 0), v100, z5, tool0;
MoveL Offs(p0,339.575,311.875, 0), v100, z5, tool0;
MoveL Offs(p0,339.01599999999996,311.3728, 0), v100, z5, tool0;
MoveL Offs(p0,338.547,310.98339999999996, 0), v100, z5, tool0;
MoveL Offs(p0,338.18,310.71760000000006, 0), v100, z5, tool0;
MoveL Offs(p0,337.927,310.5862, 0), v100, z5, tool0;
MoveL Offs(p0,337.8,310.6, 0), v100, z5, tool0;
MoveL Offs(p0,337.3896,310.3768, 0), v100, z5, tool0;
MoveL Offs(p0,337.3513,310.24089999999995, 0), v100, z5, tool0;
MoveL Offs(p0,337.3232,310.08160000000004, 0), v100, z5, tool0;
MoveL Offs(p0,337.3059,309.90070000000003, 0), v100, z5, tool0;
MoveL Offs(p0,337.3,309.7, 0), v100, z5, tool0;
MoveL Offs(p0,336.8328000000001,308.2464000000001, 0), v100, z5, tool0;
MoveL Offs(p0,336.3172,307.28709999999995, 0), v100, z5, tool0;
MoveL Offs(p0,335.6744,306.25520000000006, 0), v100, z5, tool0;
MoveL Offs(p0,334.95,305.2125, 0), v100, z5, tool0;
MoveL Offs(p0,334.1896,304.22079999999994, 0), v100, z5, tool0;
MoveL Offs(p0,333.4388,303.3419, 0), v100, z5, tool0;
MoveL Offs(p0,332.7432,302.6376, 0), v100, z5, tool0;
MoveL Offs(p0,332.14840000000004,302.16970000000003, 0), v100, z5, tool0;
MoveL Offs(p0,331.7,302.0, 0), v100, z5, tool0;
MoveL Offs(p0,331.3442,302.20520000000005, 0), v100, z5, tool0;
MoveL Offs(p0,331.1696000000001,302.78960000000006, 0), v100, z5, tool0;
MoveL Offs(p0,331.1654,303.7063999999999, 0), v100, z5, tool0;
MoveL Offs(p0,331.3208,304.90880000000004, 0), v100, z5, tool0;
MoveL Offs(p0,332.0672,307.9832, 0), v100, z5, tool0;
MoveL Offs(p0,332.6366,309.7616, 0), v100, z5, tool0;
MoveL Offs(p0,333.3224,311.6384, 0), v100, z5, tool0;
MoveL Offs(p0,334.11379999999997,313.5668, 0), v100, z5, tool0;
MoveL Offs(p0,335.0,315.5, 0), v100, z5, tool0;
MoveL Offs(p0,336.1167000000001,317.67050000000006, 0), v100, z5, tool0;
MoveL Offs(p0,337.4056000000001,319.9520000000001, 0), v100, z5, tool0;
MoveL Offs(p0,338.8349,322.29949999999997, 0), v100, z5, tool0;
MoveL Offs(p0,340.37280000000004,324.66800000000006, 0), v100, z5, tool0;
MoveL Offs(p0,341.9875,327.0125, 0), v100, z5, tool0;
MoveL Offs(p0,343.6472,329.288, 0), v100, z5, tool0;
MoveL Offs(p0,345.3201,331.4495, 0), v100, z5, tool0;
MoveL Offs(p0,346.97440000000006,333.45200000000006, 0), v100, z5, tool0;
MoveL Offs(p0,348.5783,335.2505, 0), v100, z5, tool0;
MoveL Offs(p0,350.1,336.8, 0), v100, z5, tool0;
MoveL Offs(p0,352.1322,338.6498, 0), v100, z5, tool0;
MoveL Offs(p0,355.1136000000001,341.18240000000003, 0), v100, z5, tool0;
MoveL Offs(p0,358.78139999999996,344.19259999999997, 0), v100, z5, tool0;
MoveL Offs(p0,362.8728,347.47520000000003, 0), v100, z5, tool0;
MoveL Offs(p0,367.125,350.825, 0), v100, z5, tool0;
MoveL Offs(p0,371.2751999999999,354.03679999999997, 0), v100, z5, tool0;
MoveL Offs(p0,375.0606,356.9054, 0), v100, z5, tool0;
MoveL Offs(p0,378.21840000000003,359.22560000000004, 0), v100, z5, tool0;
MoveL Offs(p0,380.48580000000004,360.7922, 0), v100, z5, tool0;
MoveL Offs(p0,381.6,361.4, 0), v100, z5, tool0;
MoveL Offs(p0,382.5696000000001,361.68640000000005, 0), v100, z5, tool0;
MoveL Offs(p0,382.8,361.8, 0), v100, z5, tool0;
MoveL Offs(p0,383.01840000000004,361.9256, 0), v100, z5, tool0;
MoveL Offs(p0,383.2212,362.06080000000003, 0), v100, z5, tool0;
MoveL Offs(p0,383.4048000000001,362.20320000000004, 0), v100, z5, tool0;
MoveL Offs(p0,383.5656,362.35040000000004, 0), v100, z5, tool0;
MoveL Offs(p0,383.7,362.5, 0), v100, z5, tool0;
MoveL Offs(p0,383.4184,362.73040000000003, 0), v100, z5, tool0;
MoveL Offs(p0,382.27690000000007,362.15510000000006, 0), v100, z5, tool0;
MoveL Offs(p0,381.96720000000005,362.08080000000007, 0), v100, z5, tool0;
MoveL Offs(p0,382.0703,362.2777, 0), v100, z5, tool0;
MoveL Offs(p0,382.5856,362.74640000000005, 0), v100, z5, tool0;
MoveL Offs(p0,383.5125,363.4875, 0), v100, z5, tool0;
MoveL Offs(p0,384.85040000000004,364.5016, 0), v100, z5, tool0;
MoveL Offs(p0,386.5987,365.78929999999997, 0), v100, z5, tool0;
MoveL Offs(p0,388.7568,367.35120000000006, 0), v100, z5, tool0;
MoveL Offs(p0,391.32410000000004,369.1879, 0), v100, z5, tool0;
MoveL Offs(p0,394.3,371.3, 0), v100, z5, tool0;
MoveL Offs(p0,396.0478000000001,372.56050000000005, 0), v100, z5, tool0;
MoveL Offs(p0,397.7344000000001,373.7520000000001, 0), v100, z5, tool0;
MoveL Offs(p0,399.33459999999997,374.85949999999997, 0), v100, z5, tool0;
MoveL Offs(p0,400.82320000000004,375.868, 0), v100, z5, tool0;
MoveL Offs(p0,402.175,376.7625, 0), v100, z5, tool0;
MoveL Offs(p0,403.3648,377.52799999999996, 0), v100, z5, tool0;
MoveL Offs(p0,404.3674,378.1495, 0), v100, z5, tool0;
MoveL Offs(p0,405.1576000000001,378.612, 0), v100, z5, tool0;
MoveL Offs(p0,405.7102,378.9005, 0), v100, z5, tool0;
MoveL Offs(p0,406.0,379.0, 0), v100, z5, tool0;
MoveL Offs(p0,406.725,379.2625, 0), v100, z5, tool0;
MoveL Offs(p0,406.8208,379.3672, 0), v100, z5, tool0;
MoveL Offs(p0,406.8974,379.4851, 0), v100, z5, tool0;
MoveL Offs(p0,406.95360000000005,379.61440000000005, 0), v100, z5, tool0;
MoveL Offs(p0,406.9882,379.7533, 0), v100, z5, tool0;
MoveL Offs(p0,407.0,379.9, 0), v100, z5, tool0;
MoveL Offs(p0,407.7168000000001,380.98320000000007, 0), v100, z5, tool0;
MoveL Offs(p0,408.50120000000004,381.6433, 0), v100, z5, tool0;
MoveL Offs(p0,409.47040000000004,382.3256, 0), v100, z5, tool0;
MoveL Offs(p0,410.55,382.9875, 0), v100, z5, tool0;
MoveL Offs(p0,411.6656,383.5864, 0), v100, z5, tool0;
MoveL Offs(p0,412.7428,384.07969999999995, 0), v100, z5, tool0;
MoveL Offs(p0,413.7072,384.42480000000006, 0), v100, z5, tool0;
MoveL Offs(p0,414.4844,384.57910000000004, 0), v100, z5, tool0;
MoveL Offs(p0,415.0,384.5, 0), v100, z5, tool0;
MoveL Offs(p0,415.8181000000001,384.8294, 0), v100, z5, tool0;
MoveL Offs(p0,415.8,385.0, 0), v100, z5, tool0;
MoveL Offs(p0,416.4928000000001,386.19440000000014, 0), v100, z5, tool0;
MoveL Offs(p0,417.4001999999999,386.93859999999995, 0), v100, z5, tool0;
MoveL Offs(p0,418.5584,387.71520000000004, 0), v100, z5, tool0;
MoveL Offs(p0,419.875,388.475, 0), v100, z5, tool0;
MoveL Offs(p0,421.2576,389.16880000000003, 0), v100, z5, tool0;
MoveL Offs(p0,422.6138000000001,389.74739999999997, 0), v100, z5, tool0;
MoveL Offs(p0,423.85120000000006,390.1616, 0), v100, z5, tool0;
MoveL Offs(p0,424.8774,390.36220000000003, 0), v100, z5, tool0;
MoveL Offs(p0,425.6,390.3, 0), v100, z5, tool0;
MoveL Offs(p0,426.0528000000001,390.01920000000007, 0), v100, z5, tool0;
MoveL Offs(p0,426.25519999999995,389.8113, 0), v100, z5, tool0;
MoveL Offs(p0,426.4384,389.5656, 0), v100, z5, tool0;
MoveL Offs(p0,426.6,389.2875, 0), v100, z5, tool0;
MoveL Offs(p0,426.73760000000004,388.9824, 0), v100, z5, tool0;
MoveL Offs(p0,426.84880000000004,388.65569999999997, 0), v100, z5, tool0;
MoveL Offs(p0,426.9312000000001,388.31280000000004, 0), v100, z5, tool0;
MoveL Offs(p0,426.98240000000004,387.95910000000003, 0), v100, z5, tool0;
MoveL Offs(p0,427.0,387.6, 0), v100, z5, tool0;
MoveL Offs(p0,427.0,387.6, 0), v100, z5, tool0;
MoveJ Offs(p0,414.9,369.9, 10), v100, z1, tool0;
MoveL Offs(p0,413.7556000000001,366.33060000000006, 0), v100, z5, tool0;
MoveL Offs(p0,412.9568000000001,362.4048000000001, 0), v100, z5, tool0;
MoveL Offs(p0,412.49519999999995,358.2162, 0), v100, z5, tool0;
MoveL Offs(p0,412.3624000000001,353.8584000000001, 0), v100, z5, tool0;
MoveL Offs(p0,412.55,349.425, 0), v100, z5, tool0;
MoveL Offs(p0,413.0496,345.0096, 0), v100, z5, tool0;
MoveL Offs(p0,413.8528,340.7058, 0), v100, z5, tool0;
MoveL Offs(p0,416.33639999999997,332.80740000000003, 0), v100, z5, tool0;
MoveL Offs(p0,418.0,329.4, 0), v100, z5, tool0;
MoveL Offs(p0,419.69710000000003,326.0556, 0), v100, z5, tool0;
MoveL Offs(p0,420.7048000000001,323.1648000000001, 0), v100, z5, tool0;
MoveL Offs(p0,420.9277,320.6411999999999, 0), v100, z5, tool0;
MoveL Offs(p0,420.2704,318.39840000000004, 0), v100, z5, tool0;
MoveL Offs(p0,418.6375,316.35, 0), v100, z5, tool0;
MoveL Offs(p0,415.93359999999996,314.4096, 0), v100, z5, tool0;
MoveL Offs(p0,412.06329999999997,312.4907999999999, 0), v100, z5, tool0;
MoveL Offs(p0,406.9312,310.5072, 0), v100, z5, tool0;
MoveL Offs(p0,400.4419,308.3724, 0), v100, z5, tool0;
MoveL Offs(p0,392.5,306.0, 0), v100, z5, tool0;
MoveL Offs(p0,388.6855,304.84380000000004, 0), v100, z5, tool0;
MoveL Offs(p0,384.7240000000001,303.4944000000001, 0), v100, z5, tool0;
MoveL Offs(p0,380.6785,301.9806, 0), v100, z5, tool0;
MoveL Offs(p0,376.61199999999997,300.3312, 0), v100, z5, tool0;
MoveL Offs(p0,372.5875,298.575, 0), v100, z5, tool0;
MoveL Offs(p0,368.668,296.74080000000004, 0), v100, z5, tool0;
MoveL Offs(p0,364.9165,294.8574, 0), v100, z5, tool0;
MoveL Offs(p0,361.396,292.9536, 0), v100, z5, tool0;
MoveL Offs(p0,358.16949999999997,291.05820000000006, 0), v100, z5, tool0;
MoveL Offs(p0,355.3,289.2, 0), v100, z5, tool0;
MoveL Offs(p0,353.88590000000005,288.2658, 0), v100, z5, tool0;
MoveL Offs(p0,352.6872000000001,287.49840000000006, 0), v100, z5, tool0;
MoveL Offs(p0,351.67929999999996,286.8906, 0), v100, z5, tool0;
MoveL Offs(p0,350.8376,286.4352, 0), v100, z5, tool0;
MoveL Offs(p0,350.1375,286.125, 0), v100, z5, tool0;
MoveL Offs(p0,349.55440000000004,285.95279999999997, 0), v100, z5, tool0;
MoveL Offs(p0,349.0637,285.9114, 0), v100, z5, tool0;
MoveL Offs(p0,348.6408,285.9936000000001, 0), v100, z5, tool0;
MoveL Offs(p0,348.2611,286.19220000000007, 0), v100, z5, tool0;
MoveL Offs(p0,347.9,286.5, 0), v100, z5, tool0;
MoveL Offs(p0,347.6049,286.71240000000006, 0), v100, z5, tool0;
MoveL Offs(p0,347.2072000000001,286.9272000000001, 0), v100, z5, tool0;
MoveL Offs(p0,346.7183,287.14079999999996, 0), v100, z5, tool0;
MoveL Offs(p0,346.1496,287.34960000000007, 0), v100, z5, tool0;
MoveL Offs(p0,345.5125,287.55, 0), v100, z5, tool0;
MoveL Offs(p0,344.8184,287.7384, 0), v100, z5, tool0;
MoveL Offs(p0,344.0786999999999,287.91119999999995, 0), v100, z5, tool0;
MoveL Offs(p0,343.3048,288.0648, 0), v100, z5, tool0;
MoveL Offs(p0,342.5081,288.1956, 0), v100, z5, tool0;
MoveL Offs(p0,341.7,288.3, 0), v100, z5, tool0;
MoveL Offs(p0,339.03200000000004,288.56000000000006, 0), v100, z5, tool0;
MoveL Offs(p0,338.1,288.70950000000005, 0), v100, z5, tool0;
MoveL Offs(p0,337.372,288.91600000000005, 0), v100, z5, tool0;
MoveL Offs(p0,336.8,289.2125, 0), v100, z5, tool0;
MoveL Offs(p0,336.336,289.632, 0), v100, z5, tool0;
MoveL Offs(p0,335.932,290.20750000000004, 0), v100, z5, tool0;
MoveL Offs(p0,335.5400000000001,290.97200000000004, 0), v100, z5, tool0;
MoveL Offs(p0,335.112,291.9585, 0), v100, z5, tool0;
MoveL Offs(p0,334.6,293.2, 0), v100, z5, tool0;
MoveL Offs(p0,334.19930000000005,294.1586000000001, 0), v100, z5, tool0;
MoveL Offs(p0,333.90240000000017,294.9648000000001, 0), v100, z5, tool0;
MoveL Offs(p0,333.71709999999996,295.6642, 0), v100, z5, tool0;
MoveL Offs(p0,333.6512,296.30240000000003, 0), v100, z5, tool0;
MoveL Offs(p0,333.7125,296.925, 0), v100, z5, tool0;
MoveL Offs(p0,333.90880000000004,297.57759999999996, 0), v100, z5, tool0;
MoveL Offs(p0,334.24789999999996,298.3058, 0), v100, z5, tool0;
MoveL Offs(p0,335.3857,300.1714, 0), v100, z5, tool0;
MoveL Offs(p0,336.2,301.4, 0), v100, z5, tool0;
MoveL Offs(p0,339.02930000000003,305.15430000000003, 0), v100, z5, tool0;
MoveL Offs(p0,343.3184000000001,310.1224, 0), v100, z5, tool0;
MoveL Offs(p0,348.7991,316.04209999999995, 0), v100, z5, tool0;
MoveL Offs(p0,355.20320000000004,322.6512, 0), v100, z5, tool0;
MoveL Offs(p0,362.2625,329.6875, 0), v100, z5, tool0;
MoveL Offs(p0,369.7088,336.8888, 0), v100, z5, tool0;
MoveL Offs(p0,377.27389999999997,343.9929, 0), v100, z5, tool0;
MoveL Offs(p0,384.68960000000004,350.73760000000004, 0), v100, z5, tool0;
MoveL Offs(p0,391.68770000000006,356.8607, 0), v100, z5, tool0;
MoveL Offs(p0,398.0,362.1, 0), v100, z5, tool0;
MoveL Offs(p0,400.8213,364.3113, 0), v100, z5, tool0;
MoveL Offs(p0,403.5544000000001,366.4224000000001, 0), v100, z5, tool0;
MoveL Offs(p0,406.1531,368.3991, 0), v100, z5, tool0;
MoveL Offs(p0,408.57120000000003,370.2072, 0), v100, z5, tool0;
MoveL Offs(p0,410.7625,371.8125, 0), v100, z5, tool0;
MoveL Offs(p0,412.6808,373.1808, 0), v100, z5, tool0;
MoveL Offs(p0,414.2799,374.27789999999993, 0), v100, z5, tool0;
MoveL Offs(p0,415.51360000000005,375.0696, 0), v100, z5, tool0;
MoveL Offs(p0,416.3357,375.5217, 0), v100, z5, tool0;
MoveL Offs(p0,416.7,375.6, 0), v100, z5, tool0;
MoveL Offs(p0,416.4696,374.4144, 0), v100, z5, tool0;
MoveL Offs(p0,416.2875,373.8375, 0), v100, z5, tool0;
MoveL Offs(p0,416.0664,373.17359999999996, 0), v100, z5, tool0;
MoveL Offs(p0,415.81170000000003,372.4353, 0), v100, z5, tool0;
MoveL Offs(p0,415.52880000000005,371.6352, 0), v100, z5, tool0;
MoveL Offs(p0,415.22310000000004,370.7859, 0), v100, z5, tool0;
MoveL Offs(p0,414.9,369.9, 0), v100, z5, tool0;
MoveL Offs(p0,414.9,369.9, 0), v100, z5, tool0;
MoveJ Offs(p0,247.4,368.0, 10), v100, z1, tool0;
MoveL Offs(p0,249.02240000000006,367.4943, 0), v100, z5, tool0;
MoveL Offs(p0,250.57520000000008,367.0024000000001, 0), v100, z5, tool0;
MoveL Offs(p0,252.03679999999994,366.5321, 0), v100, z5, tool0;
MoveL Offs(p0,253.38559999999998,366.0912000000001, 0), v100, z5, tool0;
MoveL Offs(p0,254.6,365.6875, 0), v100, z5, tool0;
MoveL Offs(p0,255.65839999999997,365.32879999999994, 0), v100, z5, tool0;
MoveL Offs(p0,256.5392,365.02290000000005, 0), v100, z5, tool0;
MoveL Offs(p0,257.2208,364.77760000000006, 0), v100, z5, tool0;
MoveL Offs(p0,257.6816,364.6007, 0), v100, z5, tool0;
MoveL Offs(p0,257.9,364.5, 0), v100, z5, tool0;
MoveL Offs(p0,257.4239,364.257, 0), v100, z5, tool0;
MoveL Offs(p0,257.0008,364.18800000000005, 0), v100, z5, tool0;
MoveL Offs(p0,256.4625,364.125, 0), v100, z5, tool0;
MoveL Offs(p0,255.8192,364.068, 0), v100, z5, tool0;
MoveL Offs(p0,255.08109999999996,364.017, 0), v100, z5, tool0;
MoveL Offs(p0,254.2584,363.97200000000004, 0), v100, z5, tool0;
MoveL Offs(p0,253.36130000000003,363.933, 0), v100, z5, tool0;
MoveL Offs(p0,252.4,363.9, 0), v100, z5, tool0;
MoveL Offs(p0,246.9375,363.6375, 0), v100, z5, tool0;
MoveL Offs(p0,245.8192,363.5328, 0), v100, z5, tool0;
MoveL Offs(p0,244.74409999999997,363.41490000000005, 0), v100, z5, tool0;
MoveL Offs(p0,243.7344,363.28560000000004, 0), v100, z5, tool0;
MoveL Offs(p0,242.8123,363.1467, 0), v100, z5, tool0;
MoveL Offs(p0,242.0,363.0, 0), v100, z5, tool0;
MoveL Offs(p0,240.3904,362.7288000000001, 0), v100, z5, tool0;
MoveL Offs(p0,239.52859999999995,362.5752, 0), v100, z5, tool0;
MoveL Offs(p0,238.65120000000007,362.41440000000006, 0), v100, z5, tool0;
MoveL Offs(p0,237.775,362.25, 0), v100, z5, tool0;
MoveL Offs(p0,236.91679999999997,362.0856, 0), v100, z5, tool0;
MoveL Offs(p0,236.09340000000003,361.92480000000006, 0), v100, z5, tool0;
MoveL Offs(p0,235.32160000000005,361.7712, 0), v100, z5, tool0;
MoveL Offs(p0,234.61819999999997,361.62840000000006, 0), v100, z5, tool0;
MoveL Offs(p0,234.0,361.5, 0), v100, z5, tool0;
MoveL Offs(p0,232.2704000000001,361.22400000000005, 0), v100, z5, tool0;
MoveL Offs(p0,231.5826,361.22099999999995, 0), v100, z5, tool0;
MoveL Offs(p0,229.7808,361.968, 0), v100, z5, tool0;
MoveL Offs(p0,229.1434,362.529, 0), v100, z5, tool0;
MoveL Offs(p0,228.42560000000003,363.276, 0), v100, z5, tool0;
MoveL Offs(p0,227.5902,364.22700000000003, 0), v100, z5, tool0;
MoveL Offs(p0,226.6,365.4, 0), v100, z5, tool0;
MoveL Offs(p0,226.0192,366.15090000000004, 0), v100, z5, tool0;
MoveL Offs(p0,225.48160000000001,366.8952000000001, 0), v100, z5, tool0;
MoveL Offs(p0,224.99439999999996,367.62029999999993, 0), v100, z5, tool0;
MoveL Offs(p0,224.56480000000002,368.31360000000006, 0), v100, z5, tool0;
MoveL Offs(p0,224.2,368.9625, 0), v100, z5, tool0;
MoveL Offs(p0,223.90719999999996,369.5544, 0), v100, z5, tool0;
MoveL Offs(p0,223.6936,370.07669999999996, 0), v100, z5, tool0;
MoveL Offs(p0,223.56640000000002,370.51680000000005, 0), v100, z5, tool0;
MoveL Offs(p0,223.5328,370.8621, 0), v100, z5, tool0;
MoveL Offs(p0,223.6,371.1, 0), v100, z5, tool0;
MoveL Offs(p0,224.2367,371.56940000000003, 0), v100, z5, tool0;
MoveL Offs(p0,225.44160000000005,371.84320000000014, 0), v100, z5, tool0;
MoveL Offs(p0,227.14690000000004,371.9298, 0), v100, z5, tool0;
MoveL Offs(p0,229.28480000000005,371.8376, 0), v100, z5, tool0;
MoveL Offs(p0,231.7875,371.575, 0), v100, z5, tool0;
MoveL Offs(p0,237.61610000000002,370.57219999999995, 0), v100, z5, tool0;
MoveL Offs(p0,240.80640000000002,369.84880000000004, 0), v100, z5, tool0;
MoveL Offs(p0,244.0903,368.9886, 0), v100, z5, tool0;
MoveL Offs(p0,247.4,368.0, 0), v100, z5, tool0;
MoveL Offs(p0,247.4,368.0, 0), v100, z5, tool0;
MoveJ Offs(p0,285.0,360.4, 10), v100, z1, tool0;
MoveL Offs(p0,284.1308,359.25270000000006, 0), v100, z5, tool0;
MoveL Offs(p0,283.2784000000001,358.2776000000001, 0), v100, z5, tool0;
MoveL Offs(p0,282.4656,357.48490000000004, 0), v100, z5, tool0;
MoveL Offs(p0,281.71520000000004,356.88480000000004, 0), v100, z5, tool0;
MoveL Offs(p0,281.05,356.4875, 0), v100, z5, tool0;
MoveL Offs(p0,280.4928,356.3032, 0), v100, z5, tool0;
MoveL Offs(p0,280.0664,356.34209999999996, 0), v100, z5, tool0;
MoveL Offs(p0,279.79359999999997,356.61440000000005, 0), v100, z5, tool0;
MoveL Offs(p0,279.69719999999995,357.13030000000003, 0), v100, z5, tool0;
MoveL Offs(p0,279.8,357.9, 0), v100, z5, tool0;
MoveL Offs(p0,279.56899999999996,358.7134, 0), v100, z5, tool0;
MoveL Offs(p0,279.46400000000006,358.7096, 0), v100, z5, tool0;
MoveL Offs(p0,279.341,358.67220000000003, 0), v100, z5, tool0;
MoveL Offs(p0,279.2,358.6, 0), v100, z5, tool0;
MoveL Offs(p0,276.75,358.95, 0), v100, z5, tool0;
MoveL Offs(p0,275.90959999999995,359.1832, 0), v100, z5, tool0;
MoveL Offs(p0,274.98879999999997,359.4596, 0), v100, z5, tool0;
MoveL Offs(p0,274.0032,359.77440000000007, 0), v100, z5, tool0;
MoveL Offs(p0,272.96840000000003,360.1228, 0), v100, z5, tool0;
MoveL Offs(p0,271.9,360.5, 0), v100, z5, tool0;
MoveL Offs(p0,265.5,362.8, 0), v100, z5, tool0;
MoveL Offs(p0,272.0,362.3, 0), v100, z5, tool0;
MoveL Offs(p0,280.46719999999993,362.7464, 0), v100, z5, tool0;
MoveL Offs(p0,281.9806,363.11619999999994, 0), v100, z5, tool0;
MoveL Offs(p0,283.67040000000003,363.5928, 0), v100, z5, tool0;
MoveL Offs(p0,285.59180000000003,364.18460000000005, 0), v100, z5, tool0;
MoveL Offs(p0,287.8,364.9, 0), v100, z5, tool0;
MoveL Offs(p0,287.3904,364.108, 0), v100, z5, tool0;
MoveL Offs(p0,287.1125,363.6625, 0), v100, z5, tool0;
MoveL Offs(p0,286.7776,363.136, 0), v100, z5, tool0;
MoveL Offs(p0,286.3923,362.5375, 0), v100, z5, tool0;
MoveL Offs(p0,285.96320000000003,361.87600000000003, 0), v100, z5, tool0;
MoveL Offs(p0,285.4969,361.1605, 0), v100, z5, tool0;
MoveL Offs(p0,285.0,360.4, 0), v100, z5, tool0;
MoveL Offs(p0,285.0,360.4, 0), v100, z5, tool0;
MoveJ Offs(p0,185.4,357.4, 10), v100, z1, tool0;
MoveL Offs(p0,185.60160000000008,356.3152000000001, 0), v100, z5, tool0;
MoveL Offs(p0,185.62589999999997,355.8088, 0), v100, z5, tool0;
MoveL Offs(p0,185.17109999999997,353.93919999999997, 0), v100, z5, tool0;
MoveL Offs(p0,184.91040000000004,353.49280000000005, 0), v100, z5, tool0;
MoveL Offs(p0,184.5873,353.0476, 0), v100, z5, tool0;
MoveL Offs(p0,184.2,352.6, 0), v100, z5, tool0;
MoveL Offs(p0,183.1467,351.32980000000003, 0), v100, z5, tool0;
MoveL Offs(p0,181.98960000000005,349.72240000000005, 0), v100, z5, tool0;
MoveL Offs(p0,180.7629,347.8426, 0), v100, z5, tool0;
MoveL Offs(p0,179.50080000000003,345.7552, 0), v100, z5, tool0;
MoveL Offs(p0,178.2375,343.525, 0), v100, z5, tool0;
MoveL Offs(p0,177.00719999999998,341.21680000000003, 0), v100, z5, tool0;
MoveL Offs(p0,175.8441,338.8954, 0), v100, z5, tool0;
MoveL Offs(p0,174.7824,336.6256, 0), v100, z5, tool0;
MoveL Offs(p0,173.8563,334.47220000000004, 0), v100, z5, tool0;
MoveL Offs(p0,173.1,332.5, 0), v100, z5, tool0;
MoveL Offs(p0,172.7321,331.3927, 0), v100, z5, tool0;
MoveL Offs(p0,172.35280000000006,330.0736000000001, 0), v100, z5, tool0;
MoveL Offs(p0,171.96869999999998,328.57689999999997, 0), v100, z5, tool0;
MoveL Offs(p0,171.58639999999997,326.93680000000006, 0), v100, z5, tool0;
MoveL Offs(p0,171.2125,325.1875, 0), v100, z5, tool0;
MoveL Offs(p0,170.8536,323.3632, 0), v100, z5, tool0;
MoveL Offs(p0,170.5163,321.49809999999997, 0), v100, z5, tool0;
MoveL Offs(p0,170.2072,319.6264, 0), v100, z5, tool0;
MoveL Offs(p0,169.9329,317.7823, 0), v100, z5, tool0;
MoveL Offs(p0,169.7,316.0, 0), v100, z5, tool0;
MoveL Offs(p0,168.5,305.5, 0), v100, z5, tool0;
MoveL Offs(p0,159.8,305.2, 0), v100, z5, tool0;
MoveL Offs(p0,151.8008,305.42319999999995, 0), v100, z5, tool0;
MoveL Offs(p0,151.3734,305.6326, 0), v100, z5, tool0;
MoveL Offs(p0,151.1056,305.91040000000004, 0), v100, z5, tool0;
MoveL Offs(p0,150.96020000000001,306.2638, 0), v100, z5, tool0;
MoveL Offs(p0,150.9,306.7, 0), v100, z5, tool0;
MoveL Offs(p0,151.17760000000004,313.8424000000001, 0), v100, z5, tool0;
MoveL Offs(p0,151.7559,317.7331, 0), v100, z5, tool0;
MoveL Offs(p0,152.5928,321.7192, 0), v100, z5, tool0;
MoveL Offs(p0,153.6625,325.7125, 0), v100, z5, tool0;
MoveL Offs(p0,154.93919999999997,329.6248, 0), v100, z5, tool0;
MoveL Offs(p0,156.3971,333.3679, 0), v100, z5, tool0;
MoveL Offs(p0,158.01040000000003,336.85360000000003, 0), v100, z5, tool0;
MoveL Offs(p0,159.7533,339.99370000000005, 0), v100, z5, tool0;
MoveL Offs(p0,161.6,342.7, 0), v100, z5, tool0;
MoveL Offs(p0,162.022,343.22390000000007, 0), v100, z5, tool0;
MoveL Offs(p0,162.44400000000005,343.7112000000001, 0), v100, z5, tool0;
MoveL Offs(p0,162.85999999999999,344.1553, 0), v100, z5, tool0;
MoveL Offs(p0,163.26399999999998,344.5496, 0), v100, z5, tool0;
MoveL Offs(p0,163.65,344.8875, 0), v100, z5, tool0;
MoveL Offs(p0,164.012,345.1624, 0), v100, z5, tool0;
MoveL Offs(p0,164.344,345.36769999999996, 0), v100, z5, tool0;
MoveL Offs(p0,164.64000000000001,345.4968, 0), v100, z5, tool0;
MoveL Offs(p0,164.894,345.5431, 0), v100, z5, tool0;
MoveL Offs(p0,165.1,345.5, 0), v100, z5, tool0;
MoveL Offs(p0,165.56199999999998,345.7177, 0), v100, z5, tool0;
MoveL Offs(p0,165.532,345.8808, 0), v100, z5, tool0;
MoveL Offs(p0,165.478,346.0751, 0), v100, z5, tool0;
MoveL Offs(p0,165.4,346.3, 0), v100, z5, tool0;
MoveL Offs(p0,165.64280000000002,347.34010000000006, 0), v100, z5, tool0;
MoveL Offs(p0,166.77840000000003,348.8608000000001, 0), v100, z5, tool0;
MoveL Offs(p0,168.6076,350.7127, 0), v100, z5, tool0;
MoveL Offs(p0,170.93120000000002,352.7464, 0), v100, z5, tool0;
MoveL Offs(p0,173.55,354.8125, 0), v100, z5, tool0;
MoveL Offs(p0,176.26479999999998,356.7616, 0), v100, z5, tool0;
MoveL Offs(p0,178.87640000000002,358.4443, 0), v100, z5, tool0;
MoveL Offs(p0,181.18560000000002,359.7112000000001, 0), v100, z5, tool0;
MoveL Offs(p0,182.9932,360.4129, 0), v100, z5, tool0;
MoveL Offs(p0,184.1,360.4, 0), v100, z5, tool0;
MoveL Offs(p0,184.36000000000007,360.1456000000002, 0), v100, z5, tool0;
MoveL Offs(p0,184.50049999999996,359.92839999999995, 0), v100, z5, tool0;
MoveL Offs(p0,184.644,359.6608, 0), v100, z5, tool0;
MoveL Offs(p0,184.7875,359.35, 0), v100, z5, tool0;
MoveL Offs(p0,184.928,359.0032, 0), v100, z5, tool0;
MoveL Offs(p0,185.0625,358.6276, 0), v100, z5, tool0;
MoveL Offs(p0,185.18800000000002,358.23040000000003, 0), v100, z5, tool0;
MoveL Offs(p0,185.30150000000003,357.8188, 0), v100, z5, tool0;
MoveL Offs(p0,185.4,357.4, 0), v100, z5, tool0;
MoveL Offs(p0,185.4,357.4, 0), v100, z5, tool0;
MoveJ Offs(p0,266.5,358.9, 10), v100, z1, tool0;
MoveL Offs(p0,267.20220000000006,358.69130000000007, 0), v100, z5, tool0;
MoveL Offs(p0,267.97760000000005,358.4304000000001, 0), v100, z5, tool0;
MoveL Offs(p0,268.8094,358.1251, 0), v100, z5, tool0;
MoveL Offs(p0,269.6808,357.7832, 0), v100, z5, tool0;
MoveL Offs(p0,270.575,357.4125, 0), v100, z5, tool0;
MoveL Offs(p0,271.4752,357.02080000000007, 0), v100, z5, tool0;
MoveL Offs(p0,272.3646,356.6159, 0), v100, z5, tool0;
MoveL Offs(p0,273.2264,356.20560000000006, 0), v100, z5, tool0;
MoveL Offs(p0,274.04380000000003,355.7977, 0), v100, z5, tool0;
MoveL Offs(p0,274.8,355.4, 0), v100, z5, tool0;
MoveL Offs(p0,279.0,352.9, 0), v100, z5, tool0;
MoveL Offs(p0,271.9,343.7, 0), v100, z5, tool0;
MoveL Offs(p0,270.7155000000001,342.1738000000001, 0), v100, z5, tool0;
MoveL Offs(p0,269.5160000000001,340.6704000000001, 0), v100, z5, tool0;
MoveL Offs(p0,268.3225,339.21259999999995, 0), v100, z5, tool0;
MoveL Offs(p0,267.15600000000006,337.82320000000004, 0), v100, z5, tool0;
MoveL Offs(p0,266.0375,336.525, 0), v100, z5, tool0;
MoveL Offs(p0,264.98799999999994,335.34080000000006, 0), v100, z5, tool0;
MoveL Offs(p0,264.0285,334.29339999999996, 0), v100, z5, tool0;
MoveL Offs(p0,263.18,333.40560000000005, 0), v100, z5, tool0;
MoveL Offs(p0,262.4635,332.7002, 0), v100, z5, tool0;
MoveL Offs(p0,261.9,332.2, 0), v100, z5, tool0;
MoveL Offs(p0,259.0,329.9, 0), v100, z5, tool0;
MoveL Offs(p0,255.3,332.9, 0), v100, z5, tool0;
MoveL Offs(p0,254.61030000000005,333.48480000000006, 0), v100, z5, tool0;
MoveL Offs(p0,253.81440000000006,334.2064000000001, 0), v100, z5, tool0;
MoveL Offs(p0,252.9321,335.04560000000004, 0), v100, z5, tool0;
MoveL Offs(p0,251.98319999999998,335.9832, 0), v100, z5, tool0;
MoveL Offs(p0,250.9875,337.0, 0), v100, z5, tool0;
MoveL Offs(p0,249.96480000000003,338.0768, 0), v100, z5, tool0;
MoveL Offs(p0,248.93489999999997,339.1944, 0), v100, z5, tool0;
MoveL Offs(p0,247.91760000000005,340.33360000000005, 0), v100, z5, tool0;
MoveL Offs(p0,246.9327,341.47520000000003, 0), v100, z5, tool0;
MoveL Offs(p0,246.0,342.6, 0), v100, z5, tool0;
MoveL Offs(p0,245.07319999999999,343.70050000000003, 0), v100, z5, tool0;
MoveL Offs(p0,244.10560000000004,344.8280000000001, 0), v100, z5, tool0;
MoveL Offs(p0,243.11639999999997,345.9615, 0), v100, z5, tool0;
MoveL Offs(p0,242.1248,347.08000000000004, 0), v100, z5, tool0;
MoveL Offs(p0,241.15,348.1625, 0), v100, z5, tool0;
MoveL Offs(p0,240.21120000000002,349.188, 0), v100, z5, tool0;
MoveL Offs(p0,239.3276,350.1355, 0), v100, z5, tool0;
MoveL Offs(p0,238.5184,350.98400000000004, 0), v100, z5, tool0;
MoveL Offs(p0,237.80280000000002,351.7125, 0), v100, z5, tool0;
MoveL Offs(p0,237.2,352.3, 0), v100, z5, tool0;
MoveL Offs(p0,236.67600000000002,352.8117, 0), v100, z5, tool0;
MoveL Offs(p0,236.18800000000005,353.3216000000001, 0), v100, z5, tool0;
MoveL Offs(p0,235.74199999999996,353.82189999999997, 0), v100, z5, tool0;
MoveL Offs(p0,235.34400000000005,354.3048, 0), v100, z5, tool0;
MoveL Offs(p0,235.0,354.7625, 0), v100, z5, tool0;
MoveL Offs(p0,234.71599999999998,355.1872, 0), v100, z5, tool0;
MoveL Offs(p0,234.498,355.5711, 0), v100, z5, tool0;
MoveL Offs(p0,234.35200000000003,355.9064, 0), v100, z5, tool0;
MoveL Offs(p0,234.28400000000002,356.1853, 0), v100, z5, tool0;
MoveL Offs(p0,234.3,356.4, 0), v100, z5, tool0;
MoveL Offs(p0,235.21779999999998,357.26110000000006, 0), v100, z5, tool0;
MoveL Offs(p0,237.22640000000007,358.03280000000007, 0), v100, z5, tool0;
MoveL Offs(p0,240.10859999999997,358.69770000000005, 0), v100, z5, tool0;
MoveL Offs(p0,243.64720000000003,359.2384, 0), v100, z5, tool0;
MoveL Offs(p0,247.625,359.6375, 0), v100, z5, tool0;
MoveL Offs(p0,251.8248,359.8776, 0), v100, z5, tool0;
MoveL Offs(p0,256.0294,359.94129999999996, 0), v100, z5, tool0;
MoveL Offs(p0,260.02160000000003,359.8112, 0), v100, z5, tool0;
MoveL Offs(p0,263.5842,359.4699, 0), v100, z5, tool0;
MoveL Offs(p0,266.5,358.9, 0), v100, z5, tool0;
MoveL Offs(p0,266.5,358.9, 0), v100, z5, tool0;
MoveJ Offs(p0,334.1,355.3, 10), v100, z1, tool0;
MoveL Offs(p0,334.3848000000001,353.3368000000001, 0), v100, z5, tool0;
MoveL Offs(p0,334.3232,352.5757, 0), v100, z5, tool0;
MoveL Offs(p0,333.6,351.2875, 0), v100, z5, tool0;
MoveL Offs(p0,332.86159999999995,350.6776, 0), v100, z5, tool0;
MoveL Offs(p0,331.82079999999996,350.0353, 0), v100, z5, tool0;
MoveL Offs(p0,330.4392,349.3192, 0), v100, z5, tool0;
MoveL Offs(p0,328.67840000000007,348.4879, 0), v100, z5, tool0;
MoveL Offs(p0,326.5,347.5, 0), v100, z5, tool0;
MoveL Offs(p0,323.55140000000006,346.2002000000001, 0), v100, z5, tool0;
MoveL Offs(p0,320.8152000000001,345.0576000000001, 0), v100, z5, tool0;
MoveL Offs(p0,318.2758,344.0674, 0), v100, z5, tool0;
MoveL Offs(p0,315.91760000000005,343.2248, 0), v100, z5, tool0;
MoveL Offs(p0,313.725,342.525, 0), v100, z5, tool0;
MoveL Offs(p0,311.68240000000003,341.9632, 0), v100, z5, tool0;
MoveL Offs(p0,309.7742,341.53459999999995, 0), v100, z5, tool0;
MoveL Offs(p0,307.9848,341.23440000000005, 0), v100, z5, tool0;
MoveL Offs(p0,306.2986,341.05780000000004, 0), v100, z5, tool0;
MoveL Offs(p0,304.7,341.0, 0), v100, z5, tool0;
MoveL Offs(p0,300.5,341.35, 0), v100, z5, tool0;
MoveL Offs(p0,300.2648,341.60479999999995, 0), v100, z5, tool0;
MoveL Offs(p0,300.1724,341.9604, 0), v100, z5, tool0;
MoveL Offs(p0,300.1976,342.4336, 0), v100, z5, tool0;
MoveL Offs(p0,300.3152,343.0412, 0), v100, z5, tool0;
MoveL Offs(p0,300.5,343.8, 0), v100, z5, tool0;
MoveL Offs(p0,300.7422,344.67500000000007, 0), v100, z5, tool0;
MoveL Offs(p0,301.04560000000004,345.4960000000001, 0), v100, z5, tool0;
MoveL Offs(p0,301.4054,346.25699999999995, 0), v100, z5, tool0;
MoveL Offs(p0,301.81680000000006,346.95200000000006, 0), v100, z5, tool0;
MoveL Offs(p0,302.275,347.575, 0), v100, z5, tool0;
MoveL Offs(p0,302.77520000000004,348.12, 0), v100, z5, tool0;
MoveL Offs(p0,303.31260000000003,348.58099999999996, 0), v100, z5, tool0;
MoveL Offs(p0,303.8824,348.95200000000006, 0), v100, z5, tool0;
MoveL Offs(p0,304.47979999999995,349.227, 0), v100, z5, tool0;
MoveL Offs(p0,305.1,349.4, 0), v100, z5, tool0;
MoveL Offs(p0,306.1008,349.7015, 0), v100, z5, tool0;
MoveL Offs(p0,306.5336,349.848, 0), v100, z5, tool0;
MoveL Offs(p0,307.0,350.0125, 0), v100, z5, tool0;
MoveL Offs(p0,307.4904,350.19199999999995, 0), v100, z5, tool0;
MoveL Offs(p0,307.9952,350.3835, 0), v100, z5, tool0;
MoveL Offs(p0,308.50480000000005,350.584, 0), v100, z5, tool0;
MoveL Offs(p0,309.0096,350.7905, 0), v100, z5, tool0;
MoveL Offs(p0,309.5,351.0, 0), v100, z5, tool0;
MoveL Offs(p0,310.03220000000005,351.20660000000004, 0), v100, z5, tool0;
MoveL Offs(p0,310.6016000000001,351.40480000000014, 0), v100, z5, tool0;
MoveL Offs(p0,311.1974,351.5922, 0), v100, z5, tool0;
MoveL Offs(p0,311.8088,351.76640000000003, 0), v100, z5, tool0;
MoveL Offs(p0,312.425,351.925, 0), v100, z5, tool0;
MoveL Offs(p0,313.0352,352.0656, 0), v100, z5, tool0;
MoveL Offs(p0,313.6286,352.18580000000003, 0), v100, z5, tool0;
MoveL Offs(p0,314.19440000000003,352.2832, 0), v100, z5, tool0;
MoveL Offs(p0,314.72180000000003,352.35540000000003, 0), v100, z5, tool0;
MoveL Offs(p0,315.2,352.4, 0), v100, z5, tool0;
MoveL Offs(p0,316.9,352.6375, 0), v100, z5, tool0;
MoveL Offs(p0,317.11519999999996,352.72400000000005, 0), v100, z5, tool0;
MoveL Offs(p0,317.2776,352.8165, 0), v100, z5, tool0;
MoveL Offs(p0,317.3824000000001,352.91200000000003, 0), v100, z5, tool0;
MoveL Offs(p0,317.42480000000006,353.0075, 0), v100, z5, tool0;
MoveL Offs(p0,317.4,353.1, 0), v100, z5, tool0;
MoveL Offs(p0,317.6333000000001,353.45660000000004, 0), v100, z5, tool0;
MoveL Offs(p0,318.5344000000001,354.00880000000006, 0), v100, z5, tool0;
MoveL Offs(p0,319.9551,354.70020000000005, 0), v100, z5, tool0;
MoveL Offs(p0,321.7472,355.4744, 0), v100, z5, tool0;
MoveL Offs(p0,323.7625,356.275, 0), v100, z5, tool0;
MoveL Offs(p0,325.8528,357.04560000000004, 0), v100, z5, tool0;
MoveL Offs(p0,327.8699,357.72979999999995, 0), v100, z5, tool0;
MoveL Offs(p0,329.6656,358.2712, 0), v100, z5, tool0;
MoveL Offs(p0,331.0917,358.6134, 0), v100, z5, tool0;
MoveL Offs(p0,332.0,358.7, 0), v100, z5, tool0;
MoveL Offs(p0,332.48720000000014,358.47120000000007, 0), v100, z5, tool0;
MoveL Offs(p0,332.73079999999993,358.2428, 0), v100, z5, tool0;
MoveL Offs(p0,332.9696,357.94960000000003, 0), v100, z5, tool0;
MoveL Offs(p0,333.2,357.6, 0), v100, z5, tool0;
MoveL Offs(p0,333.41839999999996,357.2024, 0), v100, z5, tool0;
MoveL Offs(p0,333.6212,356.7652, 0), v100, z5, tool0;
MoveL Offs(p0,333.80480000000006,356.2968, 0), v100, z5, tool0;
MoveL Offs(p0,333.9656,355.8056, 0), v100, z5, tool0;
MoveL Offs(p0,334.1,355.3, 0), v100, z5, tool0;
MoveL Offs(p0,334.1,355.3, 0), v100, z5, tool0;
MoveJ Offs(p0,195.3,352.5, 10), v100, z1, tool0;
MoveL Offs(p0,196.15680000000006,352.22880000000004, 0), v100, z5, tool0;
MoveL Offs(p0,196.54469999999998,352.07519999999994, 0), v100, z5, tool0;
MoveL Offs(p0,196.8984,351.9144, 0), v100, z5, tool0;
MoveL Offs(p0,197.2125,351.75, 0), v100, z5, tool0;
MoveL Offs(p0,197.48160000000001,351.5856, 0), v100, z5, tool0;
MoveL Offs(p0,197.70030000000003,351.4248, 0), v100, z5, tool0;
MoveL Offs(p0,197.8632,351.2712, 0), v100, z5, tool0;
MoveL Offs(p0,197.9649,351.12840000000006, 0), v100, z5, tool0;
MoveL Offs(p0,198.0,351.0, 0), v100, z5, tool0;
MoveL Offs(p0,198.2511,350.57789999999994, 0), v100, z5, tool0;
MoveL Offs(p0,198.4352,350.4208, 0), v100, z5, tool0;
MoveL Offs(p0,198.6625,350.2625, 0), v100, z5, tool0;
MoveL Offs(p0,198.9288,350.10720000000003, 0), v100, z5, tool0;
MoveL Offs(p0,199.2299,349.95910000000003, 0), v100, z5, tool0;
MoveL Offs(p0,199.56160000000003,349.8224, 0), v100, z5, tool0;
MoveL Offs(p0,199.9197,349.7013, 0), v100, z5, tool0;
MoveL Offs(p0,200.3,349.6, 0), v100, z5, tool0;
MoveL Offs(p0,201.11440000000007,349.3200000000001, 0), v100, z5, tool0;
MoveL Offs(p0,201.5771,349.114, 0), v100, z5, tool0;
MoveL Offs(p0,202.0632,348.872, 0), v100, z5, tool0;
MoveL Offs(p0,202.5625,348.6, 0), v100, z5, tool0;
MoveL Offs(p0,203.06480000000002,348.304, 0), v100, z5, tool0;
MoveL Offs(p0,203.55989999999997,347.98999999999995, 0), v100, z5, tool0;
MoveL Offs(p0,204.03760000000003,347.66400000000004, 0), v100, z5, tool0;
MoveL Offs(p0,204.48770000000002,347.332, 0), v100, z5, tool0;
MoveL Offs(p0,204.9,347.0, 0), v100, z5, tool0;
MoveL Offs(p0,205.47060000000002,346.4999, 0), v100, z5, tool0;
MoveL Offs(p0,205.92480000000006,346.0712000000001, 0), v100, z5, tool0;
MoveL Offs(p0,206.26619999999997,345.7013, 0), v100, z5, tool0;
MoveL Offs(p0,206.49840000000003,345.3776, 0), v100, z5, tool0;
MoveL Offs(p0,206.625,345.0875, 0), v100, z5, tool0;
MoveL Offs(p0,206.64960000000002,344.8184, 0), v100, z5, tool0;
MoveL Offs(p0,206.5758,344.5577, 0), v100, z5, tool0;
MoveL Offs(p0,206.40720000000002,344.2928, 0), v100, z5, tool0;
MoveL Offs(p0,206.1474,344.01110000000006, 0), v100, z5, tool0;
MoveL Offs(p0,205.8,343.7, 0), v100, z5, tool0;
MoveL Offs(p0,203.86780000000002,341.89140000000003, 0), v100, z5, tool0;
MoveL Offs(p0,202.04240000000001,339.73120000000006, 0), v100, z5, tool0;
MoveL Offs(p0,200.34059999999997,337.2578, 0), v100, z5, tool0;
MoveL Offs(p0,198.7792,334.5096, 0), v100, z5, tool0;
MoveL Offs(p0,197.375,331.525, 0), v100, z5, tool0;
MoveL Offs(p0,196.14479999999998,328.3424, 0), v100, z5, tool0;
MoveL Offs(p0,195.1054,325.0002, 0), v100, z5, tool0;
MoveL Offs(p0,194.27360000000004,321.5368, 0), v100, z5, tool0;
MoveL Offs(p0,193.6662,317.9906, 0), v100, z5, tool0;
MoveL Offs(p0,193.3,314.4, 0), v100, z5, tool0;
MoveL Offs(p0,192.7,306.3, 0), v100, z5, tool0;
MoveL Offs(p0,186.1,305.6, 0), v100, z5, tool0;
MoveL Offs(p0,182.6629,305.3381, 0), v100, z5, tool0;
MoveL Offs(p0,181.48880000000003,305.2592000000001, 0), v100, z5, tool0;
MoveL Offs(p0,180.3375,305.1875, 0), v100, z5, tool0;
MoveL Offs(p0,179.2312,305.12479999999994, 0), v100, z5, tool0;
MoveL Offs(p0,178.19209999999998,305.0729, 0), v100, z5, tool0;
MoveL Offs(p0,177.2424,305.03360000000004, 0), v100, z5, tool0;
MoveL Offs(p0,176.40429999999998,305.0087, 0), v100, z5, tool0;
MoveL Offs(p0,175.7,305.0, 0), v100, z5, tool0;
MoveL Offs(p0,172.79600000000002,305.208, 0), v100, z5, tool0;
MoveL Offs(p0,172.475,305.3875, 0), v100, z5, tool0;
MoveL Offs(p0,172.28,305.648, 0), v100, z5, tool0;
MoveL Offs(p0,172.19299999999998,306.0045, 0), v100, z5, tool0;
MoveL Offs(p0,172.196,306.47200000000004, 0), v100, z5, tool0;
MoveL Offs(p0,172.27100000000002,307.0655, 0), v100, z5, tool0;
MoveL Offs(p0,172.4,307.8, 0), v100, z5, tool0;
MoveL Offs(p0,172.62480000000008,309.0664000000001, 0), v100, z5, tool0;
MoveL Offs(p0,172.7672,309.9411, 0), v100, z5, tool0;
MoveL Offs(p0,172.9264,310.9472, 0), v100, z5, tool0;
MoveL Offs(p0,173.1,312.0625, 0), v100, z5, tool0;
MoveL Offs(p0,173.2856,313.26480000000004, 0), v100, z5, tool0;
MoveL Offs(p0,173.4808,314.53189999999995, 0), v100, z5, tool0;
MoveL Offs(p0,173.6832,315.8416, 0), v100, z5, tool0;
MoveL Offs(p0,173.8904,317.1717, 0), v100, z5, tool0;
MoveL Offs(p0,174.1,318.5, 0), v100, z5, tool0;
MoveL Offs(p0,174.49870000000004,321.0280000000001, 0), v100, z5, tool0;
MoveL Offs(p0,174.97360000000003,323.50800000000004, 0), v100, z5, tool0;
MoveL Offs(p0,175.5229,325.93399999999997, 0), v100, z5, tool0;
MoveL Offs(p0,176.14479999999998,328.3, 0), v100, z5, tool0;
MoveL Offs(p0,176.8375,330.6, 0), v100, z5, tool0;
MoveL Offs(p0,177.5992,332.82800000000003, 0), v100, z5, tool0;
MoveL Offs(p0,178.4281,334.97799999999995, 0), v100, z5, tool0;
MoveL Offs(p0,179.32240000000002,337.04400000000004, 0), v100, z5, tool0;
MoveL Offs(p0,180.28029999999998,339.02000000000004, 0), v100, z5, tool0;
MoveL Offs(p0,181.3,340.9, 0), v100, z5, tool0;
MoveL Offs(p0,182.49800000000002,342.86480000000006, 0), v100, z5, tool0;
MoveL Offs(p0,183.73200000000006,344.7744000000001, 0), v100, z5, tool0;
MoveL Offs(p0,184.972,346.5916, 0), v100, z5, tool0;
MoveL Offs(p0,186.18800000000002,348.27920000000006, 0), v100, z5, tool0;
MoveL Offs(p0,187.35,349.8, 0), v100, z5, tool0;
MoveL Offs(p0,188.42799999999997,351.1168, 0), v100, z5, tool0;
MoveL Offs(p0,189.392,352.1924, 0), v100, z5, tool0;
MoveL Offs(p0,190.21200000000005,352.98960000000005, 0), v100, z5, tool0;
MoveL Offs(p0,190.858,353.4712, 0), v100, z5, tool0;
MoveL Offs(p0,191.3,353.6, 0), v100, z5, tool0;
MoveL Offs(p0,192.1703,353.3687, 0), v100, z5, tool0;
MoveL Offs(p0,192.54960000000003,353.2704, 0), v100, z5, tool0;
MoveL Offs(p0,192.9625,353.1625, 0), v100, z5, tool0;
MoveL Offs(p0,193.4024,353.04560000000004, 0), v100, z5, tool0;
MoveL Offs(p0,193.8627,352.9203, 0), v100, z5, tool0;
MoveL Offs(p0,194.3368,352.78720000000004, 0), v100, z5, tool0;
MoveL Offs(p0,194.81810000000002,352.6469, 0), v100, z5, tool0;
MoveL Offs(p0,195.3,352.5, 0), v100, z5, tool0;
MoveL Offs(p0,195.3,352.5, 0), v100, z5, tool0;
MoveJ Offs(p0,349.4,348.5, 10), v100, z1, tool0;
MoveL Offs(p0,349.15,344.5875, 0), v100, z5, tool0;
MoveL Offs(p0,348.8384,343.76959999999997, 0), v100, z5, tool0;
MoveL Offs(p0,348.4452,342.95529999999997, 0), v100, z5, tool0;
MoveL Offs(p0,347.97280000000006,342.1512000000001, 0), v100, z5, tool0;
MoveL Offs(p0,347.4236,341.3639, 0), v100, z5, tool0;
MoveL Offs(p0,346.8,340.6, 0), v100, z5, tool0;
MoveL Offs(p0,345.8931000000001,339.3917, 0), v100, z5, tool0;
MoveL Offs(p0,344.56080000000014,337.4376000000001, 0), v100, z5, tool0;
MoveL Offs(p0,342.90569999999997,334.90389999999996, 0), v100, z5, tool0;
MoveL Offs(p0,341.0304,331.95680000000004, 0), v100, z5, tool0;
MoveL Offs(p0,339.0375,328.7625, 0), v100, z5, tool0;
MoveL Offs(p0,337.0296,325.4871999999999, 0), v100, z5, tool0;
MoveL Offs(p0,335.10929999999996,322.29709999999994, 0), v100, z5, tool0;
MoveL Offs(p0,333.3792,319.3584, 0), v100, z5, tool0;
MoveL Offs(p0,331.94190000000003,316.8373, 0), v100, z5, tool0;
MoveL Offs(p0,330.9,314.9, 0), v100, z5, tool0;
MoveL Offs(p0,329.99670000000003,312.98300000000006, 0), v100, z5, tool0;
MoveL Offs(p0,329.26560000000006,311.12000000000006, 0), v100, z5, tool0;
MoveL Offs(p0,328.7049,309.293, 0), v100, z5, tool0;
MoveL Offs(p0,328.31280000000004,307.48400000000004, 0), v100, z5, tool0;
MoveL Offs(p0,328.0875,305.675, 0), v100, z5, tool0;
MoveL Offs(p0,328.0272,303.84800000000007, 0), v100, z5, tool0;
MoveL Offs(p0,328.1301,301.985, 0), v100, z5, tool0;
MoveL Offs(p0,328.3944,300.06800000000004, 0), v100, z5, tool0;
MoveL Offs(p0,328.8183,298.079, 0), v100, z5, tool0;
MoveL Offs(p0,329.4,296.0, 0), v100, z5, tool0;
MoveL Offs(p0,330.26090000000005,293.25370000000004, 0), v100, z5, tool0;
MoveL Offs(p0,331.0312000000001,291.0336000000001, 0), v100, z5, tool0;
MoveL Offs(p0,331.78229999999996,289.2779, 0), v100, z5, tool0;
MoveL Offs(p0,332.5856,287.9248, 0), v100, z5, tool0;
MoveL Offs(p0,333.5125,286.9125, 0), v100, z5, tool0;
MoveL Offs(p0,334.6344,286.17920000000004, 0), v100, z5, tool0;
MoveL Offs(p0,336.0227,285.66310000000004, 0), v100, z5, tool0;
MoveL Offs(p0,337.7488,285.30240000000003, 0), v100, z5, tool0;
MoveL Offs(p0,339.88410000000005,285.0353, 0), v100, z5, tool0;
MoveL Offs(p0,342.5,284.8, 0), v100, z5, tool0;
MoveL Offs(p0,343.6296000000001,284.58480000000014, 0), v100, z5, tool0;
MoveL Offs(p0,344.1434,284.40669999999994, 0), v100, z5, tool0;
MoveL Offs(p0,344.6248,284.18240000000003, 0), v100, z5, tool0;
MoveL Offs(p0,345.075,283.9125, 0), v100, z5, tool0;
MoveL Offs(p0,345.4952,283.5976, 0), v100, z5, tool0;
MoveL Offs(p0,345.8866,283.2383, 0), v100, z5, tool0;
MoveL Offs(p0,346.2504,282.83520000000004, 0), v100, z5, tool0;
MoveL Offs(p0,346.5878,282.38890000000004, 0), v100, z5, tool0;
MoveL Offs(p0,346.9,281.9, 0), v100, z5, tool0;
MoveL Offs(p0,347.3499,280.93010000000004, 0), v100, z5, tool0;
MoveL Offs(p0,347.6192000000001,279.93680000000006, 0), v100, z5, tool0;
MoveL Offs(p0,347.70730000000003,278.9147, 0), v100, z5, tool0;
MoveL Offs(p0,347.6136,277.85839999999996, 0), v100, z5, tool0;
MoveL Offs(p0,347.3375,276.7625, 0), v100, z5, tool0;
MoveL Offs(p0,346.2357,274.4303, 0), v100, z5, tool0;
MoveL Offs(p0,345.40880000000004,273.18320000000006, 0), v100, z5, tool0;
MoveL Offs(p0,344.3971,271.87489999999997, 0), v100, z5, tool0;
MoveL Offs(p0,343.2,270.5, 0), v100, z5, tool0;
MoveL Offs(p0,342.34600000000006,269.5217, 0), v100, z5, tool0;
MoveL Offs(p0,341.4800000000001,268.46960000000007, 0), v100, z5, tool0;
MoveL Offs(p0,340.626,267.3779, 0), v100, z5, tool0;
MoveL Offs(p0,339.808,266.28080000000006, 0), v100, z5, tool0;
MoveL Offs(p0,339.05,265.2125, 0), v100, z5, tool0;
MoveL Offs(p0,338.376,264.20719999999994, 0), v100, z5, tool0;
MoveL Offs(p0,337.81,263.2991, 0), v100, z5, tool0;
MoveL Offs(p0,337.37600000000003,262.5224, 0), v100, z5, tool0;
MoveL Offs(p0,337.09800000000007,261.91130000000004, 0), v100, z5, tool0;
MoveL Offs(p0,337.0,261.5, 0), v100, z5, tool0;
MoveL Offs(p0,337.25600000000003,261.2472, 0), v100, z5, tool0;
MoveL Offs(p0,337.3875,261.25, 0), v100, z5, tool0;
MoveL Offs(p0,337.54,261.2768, 0), v100, z5, tool0;
MoveL Offs(p0,338.7329,261.80699999999996, 0), v100, z5, tool0;
MoveL Offs(p0,338.6381,261.327, 0), v100, z5, tool0;
MoveL Offs(p0,338.0,260.4, 0), v100, z5, tool0;
MoveL Offs(p0,337.3989,259.6132, 0), v100, z5, tool0;
MoveL Offs(p0,336.9112000000001,258.9896000000001, 0), v100, z5, tool0;
MoveL Offs(p0,336.5303,258.52439999999996, 0), v100, z5, tool0;
MoveL Offs(p0,336.2496,258.2128000000001, 0), v100, z5, tool0;
MoveL Offs(p0,336.0625,258.05, 0), v100, z5, tool0;
MoveL Offs(p0,335.9624,258.0312, 0), v100, z5, tool0;
MoveL Offs(p0,335.94269999999995,258.15160000000003, 0), v100, z5, tool0;
MoveL Offs(p0,335.9968,258.4064, 0), v100, z5, tool0;
MoveL Offs(p0,336.1181,258.79080000000005, 0), v100, z5, tool0;
MoveL Offs(p0,336.3,259.3, 0), v100, z5, tool0;
MoveL Offs(p0,336.5061,260.0641, 0), v100, z5, tool0;
MoveL Offs(p0,336.51120000000003,260.28720000000004, 0), v100, z5, tool0;
MoveL Offs(p0,336.0,261.0, 0), v100, z5, tool0;
MoveL Offs(p0,335.38880000000006,260.73760000000004, 0), v100, z5, tool0;
MoveL Offs(p0,335.275,260.6, 0), v100, z5, tool0;
MoveL Offs(p0,335.17920000000004,260.4384, 0), v100, z5, tool0;
MoveL Offs(p0,335.1026,260.2552, 0), v100, z5, tool0;
MoveL Offs(p0,335.04640000000006,260.05280000000005, 0), v100, z5, tool0;
MoveL Offs(p0,335.0118,259.83360000000005, 0), v100, z5, tool0;
MoveL Offs(p0,335.0,259.6, 0), v100, z5, tool0;
MoveL Offs(p0,334.72459999999995,258.5893, 0), v100, z5, tool0;
MoveL Offs(p0,334.52320000000003,258.1136, 0), v100, z5, tool0;
MoveL Offs(p0,334.275,257.5875, 0), v100, z5, tool0;
MoveL Offs(p0,333.9848,257.02239999999995, 0), v100, z5, tool0;
MoveL Offs(p0,333.6574,256.4297, 0), v100, z5, tool0;
MoveL Offs(p0,333.2976,255.82080000000005, 0), v100, z5, tool0;
MoveL Offs(p0,332.9102,255.2071, 0), v100, z5, tool0;
MoveL Offs(p0,332.5,254.6, 0), v100, z5, tool0;
MoveL Offs(p0,332.08990000000006,253.99570000000003, 0), v100, z5, tool0;
MoveL Offs(p0,331.70320000000004,253.38960000000006, 0), v100, z5, tool0;
MoveL Offs(p0,331.3453,252.7919, 0), v100, z5, tool0;
MoveL Offs(p0,331.02160000000003,252.21280000000002, 0), v100, z5, tool0;
MoveL Offs(p0,330.7375,251.6625, 0), v100, z5, tool0;
MoveL Offs(p0,330.49840000000006,251.15120000000002, 0), v100, z5, tool0;
MoveL Offs(p0,330.30969999999996,250.68909999999997, 0), v100, z5, tool0;
MoveL Offs(p0,330.1768,250.28640000000004, 0), v100, z5, tool0;
MoveL Offs(p0,330.1051,249.95330000000004, 0), v100, z5, tool0;
MoveL Offs(p0,330.1,249.7, 0), v100, z5, tool0;
MoveL Offs(p0,330.3625,249.425, 0), v100, z5, tool0;
MoveL Offs(p0,330.7144,249.92720000000003, 0), v100, z5, tool0;
MoveL Offs(p0,330.85330000000005,250.19140000000002, 0), v100, z5, tool0;
MoveL Offs(p0,331.0,250.5, 0), v100, z5, tool0;
MoveL Offs(p0,331.3240000000002,251.14720000000005, 0), v100, z5, tool0;
MoveL Offs(p0,331.45899999999995,251.3703, 0), v100, z5, tool0;
MoveL Offs(p0,331.576,251.5256, 0), v100, z5, tool0;
MoveL Offs(p0,331.675,251.6125, 0), v100, z5, tool0;
MoveL Offs(p0,331.756,251.6304, 0), v100, z5, tool0;
MoveL Offs(p0,331.819,251.57869999999997, 0), v100, z5, tool0;
MoveL Offs(p0,331.86400000000003,251.45680000000002, 0), v100, z5, tool0;
MoveL Offs(p0,331.891,251.2641, 0), v100, z5, tool0;
MoveL Offs(p0,331.9,251.0, 0), v100, z5, tool0;
MoveL Offs(p0,331.4914,248.4386, 0), v100, z5, tool0;
MoveL Offs(p0,331.09680000000003,248.32319999999999, 0), v100, z5, tool0;
MoveL Offs(p0,330.575,248.575, 0), v100, z5, tool0;
MoveL Offs(p0,329.92719999999997,249.19279999999998, 0), v100, z5, tool0;
MoveL Offs(p0,329.1546,250.1754, 0), v100, z5, tool0;
MoveL Offs(p0,328.2584,251.52160000000003, 0), v100, z5, tool0;
MoveL Offs(p0,327.2398,253.23020000000002, 0), v100, z5, tool0;
MoveL Offs(p0,326.1,255.3, 0), v100, z5, tool0;
MoveL Offs(p0,325.3564,256.7342, 0), v100, z5, tool0;
MoveL Offs(p0,324.51920000000007,258.3136000000001, 0), v100, z5, tool0;
MoveL Offs(p0,323.6088,260.0034, 0), v100, z5, tool0;
MoveL Offs(p0,322.64560000000006,261.7688, 0), v100, z5, tool0;
MoveL Offs(p0,321.65,263.575, 0), v100, z5, tool0;
MoveL Offs(p0,320.6424,265.3872, 0), v100, z5, tool0;
MoveL Offs(p0,319.6432,267.17060000000004, 0), v100, z5, tool0;
MoveL Offs(p0,318.67280000000005,268.89040000000006, 0), v100, z5, tool0;
MoveL Offs(p0,317.75160000000005,270.51180000000005, 0), v100, z5, tool0;
MoveL Offs(p0,316.9,272.0, 0), v100, z5, tool0;
MoveL Offs(p0,316.1007000000001,273.4005000000001, 0), v100, z5, tool0;
MoveL Offs(p0,315.3296000000001,274.7680000000001, 0), v100, z5, tool0;
MoveL Offs(p0,314.5969,276.0815, 0), v100, z5, tool0;
MoveL Offs(p0,313.91280000000006,277.32000000000005, 0), v100, z5, tool0;
MoveL Offs(p0,313.2875,278.4625, 0), v100, z5, tool0;
MoveL Offs(p0,312.73119999999994,279.48799999999994, 0), v100, z5, tool0;
MoveL Offs(p0,312.2541,280.3755, 0), v100, z5, tool0;
MoveL Offs(p0,311.86640000000006,281.104, 0), v100, z5, tool0;
MoveL Offs(p0,311.5783,281.65250000000003, 0), v100, z5, tool0;
MoveL Offs(p0,311.4,282.0, 0), v100, z5, tool0;
MoveL Offs(p0,310.59450000000004,283.40740000000005, 0), v100, z5, tool0;
MoveL Offs(p0,309.37200000000007,284.6192000000001, 0), v100, z5, tool0;
MoveL Offs(p0,307.8135,285.6198, 0), v100, z5, tool0;
MoveL Offs(p0,306.0,286.3936, 0), v100, z5, tool0;
MoveL Offs(p0,304.0125,286.925, 0), v100, z5, tool0;
MoveL Offs(p0,301.93199999999996,287.1984, 0), v100, z5, tool0;
MoveL Offs(p0,299.8395,287.1982, 0), v100, z5, tool0;
MoveL Offs(p0,297.81600000000003,286.90880000000004, 0), v100, z5, tool0;
MoveL Offs(p0,295.9425,286.31460000000004, 0), v100, z5, tool0;
MoveL Offs(p0,294.3,285.4, 0), v100, z5, tool0;
MoveL Offs(p0,293.64300000000003,284.9345, 0), v100, z5, tool0;
MoveL Offs(p0,293.0400000000001,284.5560000000001, 0), v100, z5, tool0;
MoveL Offs(p0,292.473,284.26149999999996, 0), v100, z5, tool0;
MoveL Offs(p0,291.92400000000004,284.04800000000006, 0), v100, z5, tool0;
MoveL Offs(p0,291.375,283.9125, 0), v100, z5, tool0;
MoveL Offs(p0,290.808,283.852, 0), v100, z5, tool0;
MoveL Offs(p0,290.205,283.8635, 0), v100, z5, tool0;
MoveL Offs(p0,289.54800000000006,283.9440000000001, 0), v100, z5, tool0;
MoveL Offs(p0,288.8190000000001,284.0905, 0), v100, z5, tool0;
MoveL Offs(p0,288.0,284.3, 0), v100, z5, tool0;
MoveL Offs(p0,284.5,285.2, 0), v100, z5, tool0;
MoveL Offs(p0,287.7,286.8, 0), v100, z5, tool0;
MoveL Offs(p0,288.9493,287.52220000000005, 0), v100, z5, tool0;
MoveL Offs(p0,290.11040000000014,288.47360000000015, 0), v100, z5, tool0;
MoveL Offs(p0,291.17310000000003,289.6314, 0), v100, z5, tool0;
MoveL Offs(p0,292.1272,290.97280000000006, 0), v100, z5, tool0;
MoveL Offs(p0,292.9625,292.475, 0), v100, z5, tool0;
MoveL Offs(p0,293.66880000000003,294.1152, 0), v100, z5, tool0;
MoveL Offs(p0,294.2359,295.8706, 0), v100, z5, tool0;
MoveL Offs(p0,294.6536,297.71840000000003, 0), v100, z5, tool0;
MoveL Offs(p0,294.9117,299.6358, 0), v100, z5, tool0;
MoveL Offs(p0,295.0,301.6, 0), v100, z5, tool0;
MoveL Offs(p0,294.6880000000001,305.27120000000014, 0), v100, z5, tool0;
MoveL Offs(p0,294.325,307.2583, 0), v100, z5, tool0;
MoveL Offs(p0,293.848,309.27360000000004, 0), v100, z5, tool0;
MoveL Offs(p0,293.275,311.2625, 0), v100, z5, tool0;
MoveL Offs(p0,292.62399999999997,313.1704, 0), v100, z5, tool0;
MoveL Offs(p0,291.913,314.94269999999995, 0), v100, z5, tool0;
MoveL Offs(p0,291.16,316.5248, 0), v100, z5, tool0;
MoveL Offs(p0,290.383,317.8621, 0), v100, z5, tool0;
MoveL Offs(p0,289.6,318.9, 0), v100, z5, tool0;
MoveL Offs(p0,289.11980000000005,319.4346000000001, 0), v100, z5, tool0;
MoveL Offs(p0,288.77040000000005,319.9368000000001, 0), v100, z5, tool0;
MoveL Offs(p0,288.5686,320.4642, 0), v100, z5, tool0;
MoveL Offs(p0,288.5312,321.0744000000001, 0), v100, z5, tool0;
MoveL Offs(p0,288.675,321.825, 0), v100, z5, tool0;
MoveL Offs(p0,289.0168,322.77360000000004, 0), v100, z5, tool0;
MoveL Offs(p0,290.3616,325.4952, 0), v100, z5, tool0;
MoveL Offs(p0,291.3982,327.38340000000005, 0), v100, z5, tool0;
MoveL Offs(p0,292.7,329.7, 0), v100, z5, tool0;
MoveL Offs(p0,293.6541000000001,331.3742000000001, 0), v100, z5, tool0;
MoveL Offs(p0,294.5368,332.8576000000001, 0), v100, z5, tool0;
MoveL Offs(p0,295.3487,334.1514, 0), v100, z5, tool0;
MoveL Offs(p0,296.09040000000005,335.2568, 0), v100, z5, tool0;
MoveL Offs(p0,296.7625,336.175, 0), v100, z5, tool0;
MoveL Offs(p0,297.3656,336.9072, 0), v100, z5, tool0;
MoveL Offs(p0,297.90029999999996,337.4546, 0), v100, z5, tool0;
MoveL Offs(p0,298.3672,337.8184, 0), v100, z5, tool0;
MoveL Offs(p0,298.7669,337.99980000000005, 0), v100, z5, tool0;
MoveL Offs(p0,299.1,338.0, 0), v100, z5, tool0;
MoveL Offs(p0,300.48510000000005,337.6811000000001, 0), v100, z5, tool0;
MoveL Offs(p0,302.0928,337.5008000000001, 0), v100, z5, tool0;
MoveL Offs(p0,303.8817,337.45369999999997, 0), v100, z5, tool0;
MoveL Offs(p0,305.81039999999996,337.5344, 0), v100, z5, tool0;
MoveL Offs(p0,307.8375,337.7375, 0), v100, z5, tool0;
MoveL Offs(p0,312.0213,338.4893, 0), v100, z5, tool0;
MoveL Offs(p0,314.09520000000003,339.02720000000005, 0), v100, z5, tool0;
MoveL Offs(p0,316.1019,339.6659000000001, 0), v100, z5, tool0;
MoveL Offs(p0,318.0,340.4, 0), v100, z5, tool0;
MoveL Offs(p0,319.0801000000001,340.87, 0), v100, z5, tool0;
MoveL Offs(p0,320.14880000000005,341.3160000000001, 0), v100, z5, tool0;
MoveL Offs(p0,321.18870000000004,341.73199999999997, 0), v100, z5, tool0;
MoveL Offs(p0,322.18240000000003,342.112, 0), v100, z5, tool0;
MoveL Offs(p0,323.1125,342.45, 0), v100, z5, tool0;
MoveL Offs(p0,323.9616,342.73999999999995, 0), v100, z5, tool0;
MoveL Offs(p0,324.71229999999997,342.976, 0), v100, z5, tool0;
MoveL Offs(p0,325.34720000000004,343.15200000000004, 0), v100, z5, tool0;
MoveL Offs(p0,325.84890000000007,343.262, 0), v100, z5, tool0;
MoveL Offs(p0,326.2,343.3, 0), v100, z5, tool0;
MoveL Offs(p0,327.0688,343.5448, 0), v100, z5, tool0;
MoveL Offs(p0,327.2125,343.6375, 0), v100, z5, tool0;
MoveL Offs(p0,327.3232,343.7392, 0), v100, z5, tool0;
MoveL Offs(p0,327.3991,343.8481, 0), v100, z5, tool0;
MoveL Offs(p0,327.4384,343.9624, 0), v100, z5, tool0;
MoveL Offs(p0,327.4393,344.08029999999997, 0), v100, z5, tool0;
MoveL Offs(p0,327.4,344.2, 0), v100, z5, tool0;
MoveL Offs(p0,327.6618,344.9028, 0), v100, z5, tool0;
MoveL Offs(p0,327.8192,344.9552, 0), v100, z5, tool0;
MoveL Offs(p0,327.99940000000004,344.9884, 0), v100, z5, tool0;
MoveL Offs(p0,328.2,345.0, 0), v100, z5, tool0;
MoveL Offs(p0,329.0136000000001,345.24240000000003, 0), v100, z5, tool0;
MoveL Offs(p0,329.6859,345.4896, 0), v100, z5, tool0;
MoveL Offs(p0,330.5088,345.8112, 0), v100, z5, tool0;
MoveL Offs(p0,331.4625,346.2, 0), v100, z5, tool0;
MoveL Offs(p0,332.5272,346.6488, 0), v100, z5, tool0;
MoveL Offs(p0,333.6831,347.1504, 0), v100, z5, tool0;
MoveL Offs(p0,334.91040000000004,347.6976, 0), v100, z5, tool0;
MoveL Offs(p0,336.1893,348.2832, 0), v100, z5, tool0;
MoveL Offs(p0,337.5,348.9, 0), v100, z5, tool0;
MoveL Offs(p0,339.9176000000001,350.00660000000005, 0), v100, z5, tool0;
MoveL Offs(p0,341.9728000000001,350.8648000000001, 0), v100, z5, tool0;
MoveL Offs(p0,343.6992,351.4722, 0), v100, z5, tool0;
MoveL Offs(p0,345.13040000000007,351.82640000000004, 0), v100, z5, tool0;
MoveL Offs(p0,346.3,351.925, 0), v100, z5, tool0;
MoveL Offs(p0,347.2416,351.7656, 0), v100, z5, tool0;
MoveL Offs(p0,347.98879999999997,351.34579999999994, 0), v100, z5, tool0;
MoveL Offs(p0,348.57520000000005,350.6632000000001, 0), v100, z5, tool0;
MoveL Offs(p0,349.0344,349.71540000000005, 0), v100, z5, tool0;
MoveL Offs(p0,349.4,348.5, 0), v100, z5, tool0;
MoveL Offs(p0,349.4,348.5, 0), v100, z5, tool0;
MoveJ Offs(p0,214.5,334.2, 10), v100, z1, tool0;
MoveL Offs(p0,214.75920000000002,333.3306, 0), v100, z5, tool0;
MoveL Offs(p0,214.9,333.4, 0), v100, z5, tool0;
MoveL Offs(p0,215.4221,333.0514, 0), v100, z5, tool0;
MoveL Offs(p0,216.26880000000006,331.72720000000015, 0), v100, z5, tool0;
MoveL Offs(p0,217.35070000000002,329.6398, 0), v100, z5, tool0;
MoveL Offs(p0,218.57840000000002,327.00160000000005, 0), v100, z5, tool0;
MoveL Offs(p0,219.8625,324.025, 0), v100, z5, tool0;
MoveL Offs(p0,221.1136,320.92240000000004, 0), v100, z5, tool0;
MoveL Offs(p0,222.24229999999997,317.9062, 0), v100, z5, tool0;
MoveL Offs(p0,223.15920000000006,315.1888, 0), v100, z5, tool0;
MoveL Offs(p0,223.77490000000003,312.98260000000005, 0), v100, z5, tool0;
MoveL Offs(p0,224.0,311.5, 0), v100, z5, tool0;
MoveL Offs(p0,223.50880000000006,310.99680000000006, 0), v100, z5, tool0;
MoveL Offs(p0,222.89569999999998,310.7287, 0), v100, z5, tool0;
MoveL Offs(p0,222.03840000000005,310.4504, 0), v100, z5, tool0;
MoveL Offs(p0,220.9375,310.1625, 0), v100, z5, tool0;
MoveL Offs(p0,219.59359999999998,309.86560000000003, 0), v100, z5, tool0;
MoveL Offs(p0,218.0073,309.5603, 0), v100, z5, tool0;
MoveL Offs(p0,216.17920000000004,309.2472, 0), v100, z5, tool0;
MoveL Offs(p0,214.1099,308.92690000000005, 0), v100, z5, tool0;
MoveL Offs(p0,211.8,308.6, 0), v100, z5, tool0;
MoveL Offs(p0,209.78280000000004,308.33650000000006, 0), v100, z5, tool0;
MoveL Offs(p0,207.83040000000005,308.0880000000001, 0), v100, z5, tool0;
MoveL Offs(p0,205.9716,307.85749999999996, 0), v100, z5, tool0;
MoveL Offs(p0,204.23520000000002,307.648, 0), v100, z5, tool0;
MoveL Offs(p0,202.65,307.4625, 0), v100, z5, tool0;
MoveL Offs(p0,201.2448,307.304, 0), v100, z5, tool0;
MoveL Offs(p0,200.0484,307.1755, 0), v100, z5, tool0;
MoveL Offs(p0,199.08960000000002,307.08000000000004, 0), v100, z5, tool0;
MoveL Offs(p0,198.3972,307.02049999999997, 0), v100, z5, tool0;
MoveL Offs(p0,198.0,307.0, 0), v100, z5, tool0;
MoveL Offs(p0,197.1189,307.4509, 0), v100, z5, tool0;
MoveL Offs(p0,196.9488,307.8768, 0), v100, z5, tool0;
MoveL Offs(p0,196.8375,308.4875, 0), v100, z5, tool0;
MoveL Offs(p0,196.7832,309.3112, 0), v100, z5, tool0;
MoveL Offs(p0,196.78410000000002,310.3761, 0), v100, z5, tool0;
MoveL Offs(p0,196.83840000000004,311.71040000000005, 0), v100, z5, tool0;
MoveL Offs(p0,196.94430000000003,313.3423, 0), v100, z5, tool0;
MoveL Offs(p0,197.1,315.3, 0), v100, z5, tool0;
MoveL Offs(p0,197.38020000000003,318.09630000000004, 0), v100, z5, tool0;
MoveL Offs(p0,197.80560000000008,320.7384000000001, 0), v100, z5, tool0;
MoveL Offs(p0,198.3834,323.24609999999996, 0), v100, z5, tool0;
MoveL Offs(p0,199.1208,325.6392, 0), v100, z5, tool0;
MoveL Offs(p0,200.025,327.9375, 0), v100, z5, tool0;
MoveL Offs(p0,201.1032,330.1608, 0), v100, z5, tool0;
MoveL Offs(p0,202.3626,332.3289, 0), v100, z5, tool0;
MoveL Offs(p0,203.81040000000002,334.46160000000003, 0), v100, z5, tool0;
MoveL Offs(p0,205.4538,336.5787, 0), v100, z5, tool0;
MoveL Offs(p0,207.3,338.7, 0), v100, z5, tool0;
MoveL Offs(p0,211.5,343.2, 0), v100, z5, tool0;
MoveL Offs(p0,213.2,339.4, 0), v100, z5, tool0;
MoveL Offs(p0,213.48480000000004,338.73870000000005, 0), v100, z5, tool0;
MoveL Offs(p0,213.73840000000004,338.0816000000001, 0), v100, z5, tool0;
MoveL Offs(p0,213.95959999999997,337.4389, 0), v100, z5, tool0;
MoveL Offs(p0,214.14720000000005,336.8208, 0), v100, z5, tool0;
MoveL Offs(p0,214.3,336.2375, 0), v100, z5, tool0;
MoveL Offs(p0,214.41680000000002,335.6992, 0), v100, z5, tool0;
MoveL Offs(p0,214.4964,335.2161, 0), v100, z5, tool0;
MoveL Offs(p0,214.53760000000003,334.7984, 0), v100, z5, tool0;
MoveL Offs(p0,214.5392,334.4563, 0), v100, z5, tool0;
MoveL Offs(p0,214.5,334.2, 0), v100, z5, tool0;
MoveL Offs(p0,214.5,334.2, 0), v100, z5, tool0;
MoveJ Offs(p0,289.8,311.9, 10), v100, z1, tool0;
MoveL Offs(p0,290.8711,309.33910000000003, 0), v100, z5, tool0;
MoveL Offs(p0,291.5768000000001,306.48480000000006, 0), v100, z5, tool0;
MoveL Offs(p0,291.93569999999994,303.4697, 0), v100, z5, tool0;
MoveL Offs(p0,291.9664,300.4264, 0), v100, z5, tool0;
MoveL Offs(p0,291.6875,297.4875, 0), v100, z5, tool0;
MoveL Offs(p0,291.11760000000004,294.7856, 0), v100, z5, tool0;
MoveL Offs(p0,290.27529999999996,292.4533, 0), v100, z5, tool0;
MoveL Offs(p0,289.17920000000004,290.6232, 0), v100, z5, tool0;
MoveL Offs(p0,287.84790000000004,289.4279, 0), v100, z5, tool0;
MoveL Offs(p0,286.3,289.0, 0), v100, z5, tool0;
MoveL Offs(p0,285.54,289.34560000000005, 0), v100, z5, tool0;
MoveL Offs(p0,285.3875,289.525, 0), v100, z5, tool0;
MoveL Offs(p0,285.256,289.73439999999994, 0), v100, z5, tool0;
MoveL Offs(p0,285.14849999999996,289.97020000000003, 0), v100, z5, tool0;
MoveL Offs(p0,285.06800000000004,290.22880000000004, 0), v100, z5, tool0;
MoveL Offs(p0,285.01750000000004,290.50660000000005, 0), v100, z5, tool0;
MoveL Offs(p0,285.0,290.8, 0), v100, z5, tool0;
MoveL Offs(p0,284.62469999999996,292.2292, 0), v100, z5, tool0;
MoveL Offs(p0,284.35040000000004,292.90240000000006, 0), v100, z5, tool0;
MoveL Offs(p0,284.0125,293.65, 0), v100, z5, tool0;
MoveL Offs(p0,283.6176,294.4576, 0), v100, z5, tool0;
MoveL Offs(p0,283.1723,295.31080000000003, 0), v100, z5, tool0;
MoveL Offs(p0,282.68320000000006,296.1952, 0), v100, z5, tool0;
MoveL Offs(p0,282.15690000000006,297.0964, 0), v100, z5, tool0;
MoveL Offs(p0,281.6,298.0, 0), v100, z5, tool0;
MoveL Offs(p0,278.1,303.5, 0), v100, z5, tool0;
MoveL Offs(p0,281.7,310.3, 0), v100, z5, tool0;
MoveL Offs(p0,282.3013,311.38370000000003, 0), v100, z5, tool0;
MoveL Offs(p0,282.89840000000004,312.4056000000001, 0), v100, z5, tool0;
MoveL Offs(p0,283.4811,313.3519, 0), v100, z5, tool0;
MoveL Offs(p0,284.0392,314.2088, 0), v100, z5, tool0;
MoveL Offs(p0,284.5625,314.9625, 0), v100, z5, tool0;
MoveL Offs(p0,285.0408,315.5992, 0), v100, z5, tool0;
MoveL Offs(p0,285.4639,316.10509999999994, 0), v100, z5, tool0;
MoveL Offs(p0,285.82160000000005,316.4664, 0), v100, z5, tool0;
MoveL Offs(p0,286.1037,316.6693, 0), v100, z5, tool0;
MoveL Offs(p0,286.3,316.7, 0), v100, z5, tool0;
MoveL Offs(p0,286.7696000000001,316.3640000000001, 0), v100, z5, tool0;
MoveL Offs(p0,287.07489999999996,316.0475, 0), v100, z5, tool0;
MoveL Offs(p0,287.4168,315.644, 0), v100, z5, tool0;
MoveL Offs(p0,287.7875,315.1625, 0), v100, z5, tool0;
MoveL Offs(p0,288.1792,314.61199999999997, 0), v100, z5, tool0;
MoveL Offs(p0,288.5841,314.00149999999996, 0), v100, z5, tool0;
MoveL Offs(p0,288.9944,313.34000000000003, 0), v100, z5, tool0;
MoveL Offs(p0,289.4023,312.63649999999996, 0), v100, z5, tool0;
MoveL Offs(p0,289.8,311.9, 0), v100, z5, tool0;
MoveL Offs(p0,289.8,311.9, 0), v100, z5, tool0;
MoveJ Offs(p0,49.5,303.0, 10), v100, z1, tool0;
MoveL Offs(p0,49.717699999999994,302.4596, 0), v100, z5, tool0;
MoveL Offs(p0,49.88080000000001,302.4784000000001, 0), v100, z5, tool0;
MoveL Offs(p0,50.075100000000006,302.5248, 0), v100, z5, tool0;
MoveL Offs(p0,50.3,302.6, 0), v100, z5, tool0;
MoveL Offs(p0,51.4952,302.39520000000005, 0), v100, z5, tool0;
MoveL Offs(p0,51.7625,302.125, 0), v100, z5, tool0;
MoveL Offs(p0,52.020799999999994,301.7648, 0), v100, z5, tool0;
MoveL Offs(p0,52.2719,301.3134, 0), v100, z5, tool0;
MoveL Offs(p0,52.5176,300.7696, 0), v100, z5, tool0;
MoveL Offs(p0,52.759699999999995,300.1322, 0), v100, z5, tool0;
MoveL Offs(p0,53.0,299.4, 0), v100, z5, tool0;
MoveL Offs(p0,53.32890000000001,298.3996, 0), v100, z5, tool0;
MoveL Offs(p0,53.60320000000003,297.61280000000005, 0), v100, z5, tool0;
MoveL Offs(p0,53.8343,297.0312, 0), v100, z5, tool0;
MoveL Offs(p0,54.0336,296.6464, 0), v100, z5, tool0;
MoveL Offs(p0,54.2125,296.45, 0), v100, z5, tool0;
MoveL Offs(p0,54.3824,296.43359999999996, 0), v100, z5, tool0;
MoveL Offs(p0,54.554700000000004,296.5888, 0), v100, z5, tool0;
MoveL Offs(p0,54.740800000000014,296.9072, 0), v100, z5, tool0;
MoveL Offs(p0,54.95210000000001,297.3804, 0), v100, z5, tool0;
MoveL Offs(p0,55.2,298.0, 0), v100, z5, tool0;
MoveL Offs(p0,56.1,300.4, 0), v100, z5, tool0;
MoveL Offs(p0,57.6,298.2, 0), v100, z5, tool0;
MoveL Offs(p0,57.8276,297.83209999999997, 0), v100, z5, tool0;
MoveL Offs(p0,58.02880000000001,297.4528, 0), v100, z5, tool0;
MoveL Offs(p0,58.20120000000001,297.0686999999999, 0), v100, z5, tool0;
MoveL Offs(p0,58.3424,296.6864, 0), v100, z5, tool0;
MoveL Offs(p0,58.45,296.3125, 0), v100, z5, tool0;
MoveL Offs(p0,58.52159999999999,295.9536, 0), v100, z5, tool0;
MoveL Offs(p0,58.5548,295.61629999999997, 0), v100, z5, tool0;
MoveL Offs(p0,58.54720000000001,295.3072, 0), v100, z5, tool0;
MoveL Offs(p0,58.49640000000001,295.0329, 0), v100, z5, tool0;
MoveL Offs(p0,58.4,294.8, 0), v100, z5, tool0;
MoveL Offs(p0,58.175,294.37070000000006, 0), v100, z5, tool0;
MoveL Offs(p0,58.160000000000004,294.27840000000003, 0), v100, z5, tool0;
MoveL Offs(p0,58.175,294.2125, 0), v100, z5, tool0;
MoveL Offs(p0,58.7,294.3, 0), v100, z5, tool0;
MoveL Offs(p0,59.7881,293.7474, 0), v100, z5, tool0;
MoveL Offs(p0,60.11120000000001,293.16880000000003, 0), v100, z5, tool0;
MoveL Offs(p0,60.3875,292.475, 0), v100, z5, tool0;
MoveL Offs(p0,60.60080000000001,291.7152, 0), v100, z5, tool0;
MoveL Offs(p0,60.734899999999996,290.93859999999995, 0), v100, z5, tool0;
MoveL Offs(p0,60.77360000000001,290.19440000000003, 0), v100, z5, tool0;
MoveL Offs(p0,60.700700000000005,289.53180000000003, 0), v100, z5, tool0;
MoveL Offs(p0,60.5,289.0, 0), v100, z5, tool0;
MoveL Offs(p0,60.832100000000004,287.8714, 0), v100, z5, tool0;
MoveL Offs(p0,61.0,287.8, 0), v100, z5, tool0;
MoveL Offs(p0,62.0018,286.50630000000007, 0), v100, z5, tool0;
MoveL Offs(p0,62.786400000000015,283.55840000000006, 0), v100, z5, tool0;
MoveL Offs(p0,63.352599999999995,279.27609999999993, 0), v100, z5, tool0;
MoveL Offs(p0,63.699200000000005,273.9792, 0), v100, z5, tool0;
MoveL Offs(p0,63.825,267.9875, 0), v100, z5, tool0;
MoveL Offs(p0,63.7288,261.6208, 0), v100, z5, tool0;
MoveL Offs(p0,63.409400000000005,255.1989, 0), v100, z5, tool0;
MoveL Offs(p0,62.86559999999999,249.04160000000002, 0), v100, z5, tool0;
MoveL Offs(p0,62.096199999999996,243.46870000000004, 0), v100, z5, tool0;
MoveL Offs(p0,60.76220000000001,237.53160000000003, 0), v100, z5, tool0;
MoveL Offs(p0,60.41360000000001,236.26080000000007, 0), v100, z5, tool0;
MoveL Offs(p0,60.061400000000006,235.00920000000002, 0), v100, z5, tool0;
MoveL Offs(p0,59.7128,233.79840000000004, 0), v100, z5, tool0;
MoveL Offs(p0,59.375,232.65, 0), v100, z5, tool0;
MoveL Offs(p0,59.0552,231.58559999999997, 0), v100, z5, tool0;
MoveL Offs(p0,58.7606,230.6268, 0), v100, z5, tool0;
MoveL Offs(p0,58.498400000000004,229.79520000000002, 0), v100, z5, tool0;
MoveL Offs(p0,58.275800000000004,229.11239999999998, 0), v100, z5, tool0;
MoveL Offs(p0,58.1,228.6, 0), v100, z5, tool0;
MoveL Offs(p0,57.1,226.1, 0), v100, z5, tool0;
MoveL Offs(p0,52.1,228.3, 0), v100, z5, tool0;
MoveL Offs(p0,50.839400000000005,228.85909999999998, 0), v100, z5, tool0;
MoveL Offs(p0,49.80320000000002,229.35280000000006, 0), v100, z5, tool0;
MoveL Offs(p0,48.96979999999999,229.80570000000003, 0), v100, z5, tool0;
MoveL Offs(p0,48.3176,230.2424, 0), v100, z5, tool0;
MoveL Offs(p0,47.825,230.6875, 0), v100, z5, tool0;
MoveL Offs(p0,47.4704,231.16559999999998, 0), v100, z5, tool0;
MoveL Offs(p0,47.2322,231.7013, 0), v100, z5, tool0;
MoveL Offs(p0,47.088800000000006,232.3192, 0), v100, z5, tool0;
MoveL Offs(p0,47.018600000000006,233.04390000000004, 0), v100, z5, tool0;
MoveL Offs(p0,47.0,233.9, 0), v100, z5, tool0;
MoveL Offs(p0,47.304,237.59120000000001, 0), v100, z5, tool0;
MoveL Offs(p0,47.4625,238.85, 0), v100, z5, tool0;
MoveL Offs(p0,47.647999999999996,240.19279999999998, 0), v100, z5, tool0;
MoveL Offs(p0,47.8575,241.5944, 0), v100, z5, tool0;
MoveL Offs(p0,48.08800000000001,243.02960000000002, 0), v100, z5, tool0;
MoveL Offs(p0,48.3365,244.4732, 0), v100, z5, tool0;
MoveL Offs(p0,48.6,245.9, 0), v100, z5, tool0;
MoveL Offs(p0,49.28,250.42710000000002, 0), v100, z5, tool0;
MoveL Offs(p0,49.708000000000006,255.54880000000003, 0), v100, z5, tool0;
MoveL Offs(p0,49.896,261.0857, 0), v100, z5, tool0;
MoveL Offs(p0,49.856,266.85839999999996, 0), v100, z5, tool0;
MoveL Offs(p0,49.6,272.6875, 0), v100, z5, tool0;
MoveL Offs(p0,49.14,278.3936, 0), v100, z5, tool0;
MoveL Offs(p0,47.656000000000006,288.71920000000006, 0), v100, z5, tool0;
MoveL Offs(p0,46.656000000000006,292.9799, 0), v100, z5, tool0;
MoveL Offs(p0,45.5,296.4, 0), v100, z5, tool0;
MoveL Offs(p0,45.19440000000001,297.1864000000001, 0), v100, z5, tool0;
MoveL Offs(p0,45.1346,297.4566, 0), v100, z5, tool0;
MoveL Offs(p0,45.14320000000001,297.6512, 0), v100, z5, tool0;
MoveL Offs(p0,45.225,297.775, 0), v100, z5, tool0;
MoveL Offs(p0,45.9576,297.76959999999997, 0), v100, z5, tool0;
MoveL Offs(p0,46.3802,297.65819999999997, 0), v100, z5, tool0;
MoveL Offs(p0,46.9,297.5, 0), v100, z5, tool0;
MoveL Offs(p0,47.85520000000001,297.2408000000001, 0), v100, z5, tool0;
MoveL Offs(p0,48.202299999999994,297.1922, 0), v100, z5, tool0;
MoveL Offs(p0,48.4696,297.2024, 0), v100, z5, tool0;
MoveL Offs(p0,48.6625,297.275, 0), v100, z5, tool0;
